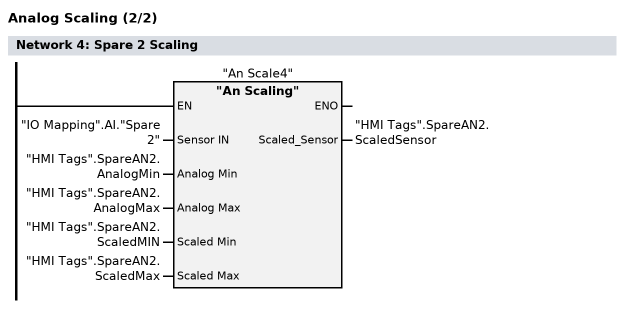
   RUNG wire#powerrail
      "An Scale4"("Sensor IN" := "IO Mapping".AI."Spare 2", "Analog Min" := "HMI Tags".SpareAN2.AnalogMin, "Analog Max" := "HMI Tags".SpareAN2.AnalogMax, "Scaled Min" := "HMI Tags".SpareAN2.ScaledMIN, "Scaled Max" := "HMI Tags".SpareAN2.ScaledMax, Scaled_Sensor => "HMI Tags".SpareAN2.ScaledSensor)
   END_RUNG
   // the same network as SCL:
   "An Scale4"("Sensor IN" := "IO Mapping".AI."Spare 2",   // "An Scaling"
               "Analog Min" := "HMI Tags".SpareAN2.AnalogMin,
               "Analog Max" := "HMI Tags".SpareAN2.AnalogMax,
               "Scaled Min" := "HMI Tags".SpareAN2.ScaledMIN,
               "Scaled Max" := "HMI Tags".SpareAN2.ScaledMax,
               Scaled_Sensor => "HMI Tags".SpareAN2.ScaledSensor);
END_REGION
END_FUNCTION

FUNCTION_BLOCK "An Scaling"   // FB5, LAD
{ S7_Optimized_Access := 'TRUE' }
// stored: MemoryReserve 100, SetENOAutomatically false
   VAR_INPUT
      "Sensor IN" : Int;
      "Analog Min" { ExternalAccessible := 'False'; ExternalVisible := 'False'; ExternalWritable := 'False'} : Int;
      "Analog Max" { ExternalAccessible := 'False'; ExternalVisible := 'False'; ExternalWritable := 'False'} : Int;
      "Scaled Min" { ExternalAccessible := 'False'; ExternalVisible := 'False'; ExternalWritable := 'False'} : Real;
      "Scaled Max" { ExternalAccessible := 'False'; ExternalVisible := 'False'; ExternalWritable := 'False'} : Real;
   END_VAR
   VAR_OUTPUT
      Scaled_Sensor : Real;
   END_VAR
   VAR
      Normalised_sensor { ExternalAccessible := 'False'; ExternalVisible := 'False'; ExternalWritable := 'False'} : Real;
      sensor_result { ExternalAccessible := 'False'; ExternalVisible := 'False'; ExternalWritable := 'False'} : Int;
   END_VAR
BEGIN

REGION Network 1: scale the sensor
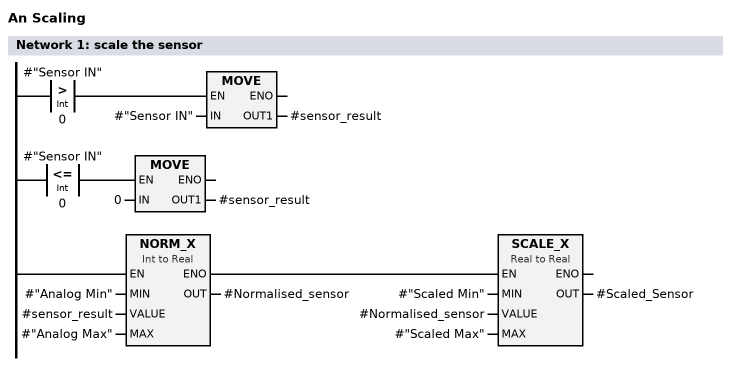
   RUNG wire#powerrail
      { S7_Templates := "SrcType := Int" } GT_Contact(in1 := #"Sensor IN", in2 := 0)
      { S7_GenerateENO := "TRUE" } Move(in := #"Sensor IN", out1 => #sensor_result)
   END_RUNG
   RUNG wire#powerrail
      { S7_Templates := "SrcType := Int" } LE_Contact(in1 := #"Sensor IN", in2 := 0)
      { S7_GenerateENO := "TRUE" } Move(in := 0, out1 => #sensor_result)
   END_RUNG
   RUNG wire#powerrail
      { S7_Templates := "[SrcType := Int, DestType := Real]"; S7_GenerateENO := "TRUE" } Normalize(min := #"Analog Min", value := #sensor_result, max := #"Analog Max", out => #Normalised_sensor)
      { S7_Templates := "[SrcType := Real, DestType := Real]"; S7_GenerateENO := "TRUE" } Scale(min := #"Scaled Min", value := #Normalised_sensor, max := #"Scaled Max", out => #Scaled_Sensor)
   END_RUNG
   // the same network as SCL:
   // ENO of a box is taken as its EN; it also drops when the box reports an error
   IF #"Sensor IN" > 0 THEN #sensor_result := #"Sensor IN"; END_IF;
   IF #"Sensor IN" <= 0 THEN #sensor_result := 0; END_IF;
   #Normalised_sensor := NORM_X(MIN := #"Analog Min", VALUE := #sensor_result, MAX := #"Analog Max");
   #Scaled_Sensor := SCALE_X(MIN := #"Scaled Min", VALUE := #Normalised_sensor, MAX := #"Scaled Max");
END_REGION
END_FUNCTION_BLOCK

FUNCTION "VFD Control" : Void   // FC9, LAD
{ S7_Optimized_Access := 'TRUE' }
// stored: SetENOAutomatically false
   VAR_TEMP   // added for the SCL form of the ladder/FBD networks
      _w1 : Bool;
   END_VAR
BEGIN

REGION Network 1: Liquids Pump
   // Refspeed = p2000, ref_Current = P2002, Ref_torque = P2003
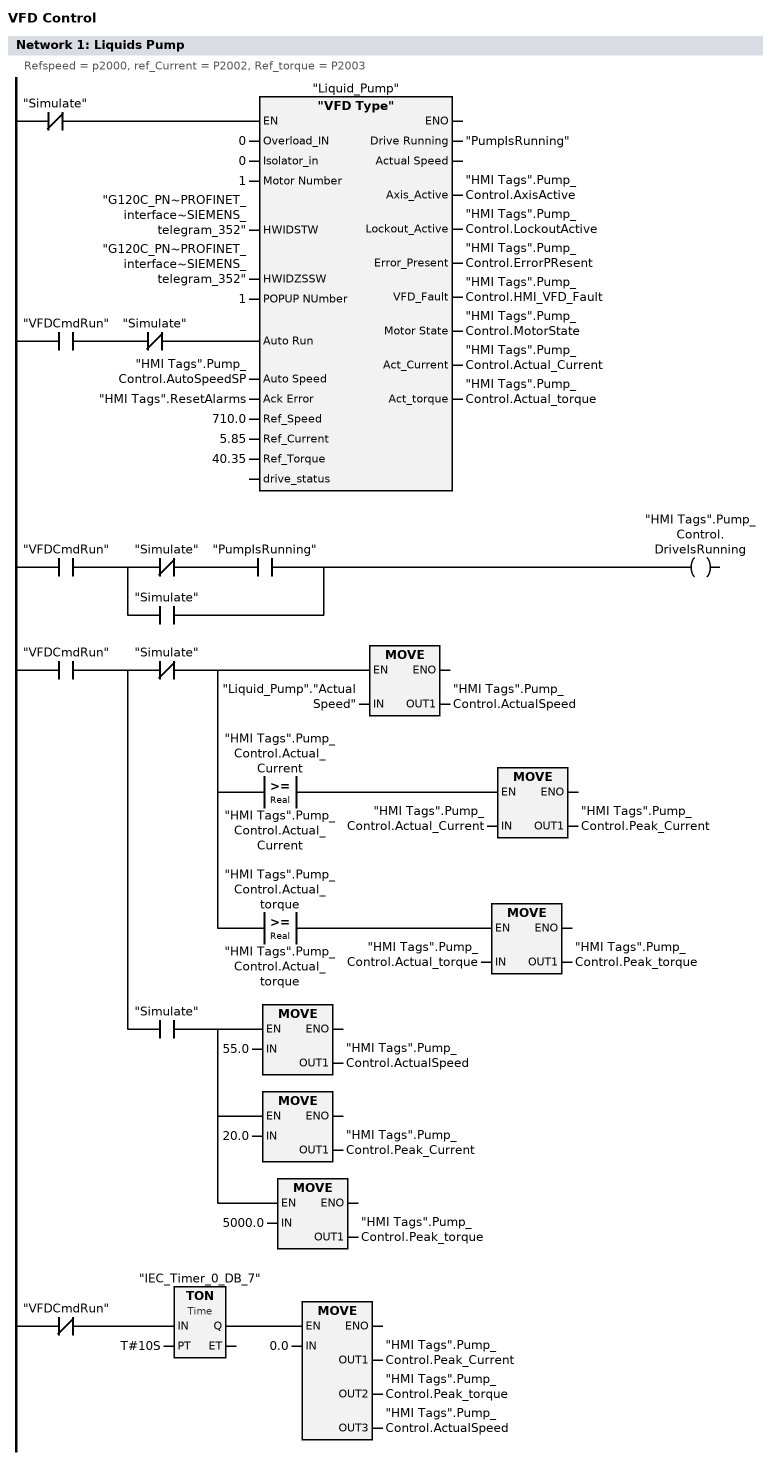
   RUNG wire#powerrail
      I_Contact( "Simulate" )
      "Liquid_Pump"("Auto Run" := wire#w1, Overload_IN := 0, Isolator_in := 0, "Motor Number" := 1, HWIDSTW := "G120C_PN~PROFINET_interface~SIEMENS_telegram_352", HWIDZSSW := "G120C_PN~PROFINET_interface~SIEMENS_telegram_352", "POPUP NUmber" := 1, "Auto Speed" := "HMI Tags".Pump_Control.AutoSpeedSP, "Ack Error" := "HMI Tags".ResetAlarms, Ref_Speed := 710.0, Ref_Current := 5.85, Ref_Torque := 40.35, drive_status :=, "Drive Running" => "PumpIsRunning", "Actual Speed" =>, Axis_Active => "HMI Tags".Pump_Control.AxisActive, Lockout_Active => "HMI Tags".Pump_Control.LockoutActive, Error_Present => "HMI Tags".Pump_Control.ErrorPResent, VFD_Fault => "HMI Tags".Pump_Control.HMI_VFD_Fault, "Motor State" => "HMI Tags".Pump_Control.MotorState, Act_Current => "HMI Tags".Pump_Control.Actual_Current, Act_torque => "HMI Tags".Pump_Control.Actual_torque)
   END_RUNG
   RUNG wire#powerrail
      Contact( "VFDCmdRun" )
      I_Contact( "Simulate" )
   END_RUNG wire#w1
   RUNG wire#powerrail
      Contact( "VFDCmdRun" )
      wire#w2
      I_Contact( "Simulate" )
      Contact( "PumpIsRunning" )
      wire#w3
      Coil( "HMI Tags".Pump_Control.DriveIsRunning )
   END_RUNG
   RUNG wire#w2
      Contact( "Simulate" )
   END_RUNG wire#w3
   RUNG wire#powerrail
      Contact( "VFDCmdRun" )
      wire#w4
      I_Contact( "Simulate" )
      wire#w5
      Move(in := "Liquid_Pump"."Actual Speed", out1 => "HMI Tags".Pump_Control.ActualSpeed)
   END_RUNG
   RUNG wire#w5
      { S7_Templates := "SrcType := Real" } GE_Contact(in1 := "HMI Tags".Pump_Control.Actual_Current, in2 := "HMI Tags".Pump_Control.Actual_Current)
      Move(in := "HMI Tags".Pump_Control.Actual_Current, out1 => "HMI Tags".Pump_Control.Peak_Current)
   END_RUNG
   RUNG wire#w5
      { S7_Templates := "SrcType := Real" } GE_Contact(in1 := "HMI Tags".Pump_Control.Actual_torque, in2 := "HMI Tags".Pump_Control.Actual_torque)
      Move(in := "HMI Tags".Pump_Control.Actual_torque, out1 => "HMI Tags".Pump_Control.Peak_torque)
   END_RUNG
   RUNG wire#w4
      Contact( "Simulate" )
      wire#w6
      Move(in := 55.0, out1 => "HMI Tags".Pump_Control.ActualSpeed)
   END_RUNG
   RUNG wire#w6
      Move(in := 20.0, out1 => "HMI Tags".Pump_Control.Peak_Current)
   END_RUNG
   RUNG wire#w6
      Move(in := 5000.0, out1 => "HMI Tags".Pump_Control.Peak_torque)
   END_RUNG
   RUNG wire#powerrail
      I_Contact( "VFDCmdRun" )
      { S7_Templates := "time_type := Time" } "IEC_Timer_0_DB_7".TON(pt := T#10S, et =>)
      Move(in := 0.0, out1 => "HMI Tags".Pump_Control.Peak_Current, out2 => "HMI Tags".Pump_Control.Peak_torque, out3 => "HMI Tags".Pump_Control.ActualSpeed)
   END_RUNG
   // the same network as SCL:
   IF NOT "Simulate" THEN
       "Liquid_Pump"(Overload_IN := 0,   // "VFD Type"
                     Isolator_in := 0,
                     "Motor Number" := 1,
                     HWIDSTW := "G120C_PN~PROFINET_interface~SIEMENS_telegram_352",
                     HWIDZSSW := "G120C_PN~PROFINET_interface~SIEMENS_telegram_352",
                     "POPUP NUmber" := 1,
                     "Auto Run" := "VFDCmdRun" AND NOT "Simulate",
                     "Auto Speed" := "HMI Tags".Pump_Control.AutoSpeedSP,
                     "Ack Error" := "HMI Tags".ResetAlarms,
                     Ref_Speed := 710.0,
                     Ref_Current := 5.85,
                     Ref_Torque := 40.35,
                     "Drive Running" => "PumpIsRunning",
                     Axis_Active => "HMI Tags".Pump_Control.AxisActive,
                     Lockout_Active => "HMI Tags".Pump_Control.LockoutActive,
                     Error_Present => "HMI Tags".Pump_Control.ErrorPResent,
                     VFD_Fault => "HMI Tags".Pump_Control.HMI_VFD_Fault,
                     "Motor State" => "HMI Tags".Pump_Control.MotorState,
                     Act_Current => "HMI Tags".Pump_Control.Actual_Current,
                     Act_torque => "HMI Tags".Pump_Control.Actual_torque);
   END_IF;
   "HMI Tags".Pump_Control.DriveIsRunning := "VFDCmdRun" AND ((NOT "Simulate" AND "PumpIsRunning") OR "Simulate");
   #_w1 := "VFDCmdRun" AND NOT "Simulate";
   IF #_w1 THEN "HMI Tags".Pump_Control.ActualSpeed := "Liquid_Pump"."Actual Speed"; END_IF;
   IF #_w1 AND ("HMI Tags".Pump_Control.Actual_Current >= "HMI Tags".Pump_Control.Actual_Current) THEN
       "HMI Tags".Pump_Control.Peak_Current := "HMI Tags".Pump_Control.Actual_Current;
   END_IF;
   IF #_w1 AND ("HMI Tags".Pump_Control.Actual_torque >= "HMI Tags".Pump_Control.Actual_torque) THEN
       "HMI Tags".Pump_Control.Peak_torque := "HMI Tags".Pump_Control.Actual_torque;
   END_IF;
   IF "VFDCmdRun" AND "Simulate" THEN
       "HMI Tags".Pump_Control.ActualSpeed := 55.0;
       "HMI Tags".Pump_Control.Peak_Current := 20.0;
       "HMI Tags".Pump_Control.Peak_torque := 5000.0;
   END_IF;
   "IEC_Timer_0_DB_7".TON(IN := NOT "VFDCmdRun", PT := T#10S);
   IF "IEC_Timer_0_DB_7".Q THEN
       "HMI Tags".Pump_Control.Peak_Current := 0.0;
       "HMI Tags".Pump_Control.Peak_torque := 0.0;
       "HMI Tags".Pump_Control.ActualSpeed := 0.0;
   END_IF;
END_REGION
END_FUNCTION

FUNCTION_BLOCK "VFD Type"   // FB9, LAD
{ S7_Optimized_Access := 'TRUE' }
// stored: MemoryReserve 100, SetENOAutomatically false
   VAR_INPUT
      Overload_IN { ExternalAccessible := 'False'; ExternalVisible := 'False'; ExternalWritable := 'False'} : Bool;
      Isolator_in { ExternalAccessible := 'False'; ExternalVisible := 'False'; ExternalWritable := 'False'} : Bool;
      "Motor Number" : Int;
      HWIDSTW { ExternalAccessible := 'False'; ExternalVisible := 'False'; ExternalWritable := 'False'} : HW_IO;
      HWIDZSSW { ExternalAccessible := 'False'; ExternalVisible := 'False'; ExternalWritable := 'False'} : HW_IO;
      "POPUP NUmber" : Int;
      "Auto Run" : Bool;
      "Auto Speed" : Real;
      "Ack Error" : Bool;
      Ref_Speed { ExternalAccessible := 'False'; ExternalVisible := 'False'; ExternalWritable := 'False'} : Real;
      Ref_Current : Real;
      Ref_Torque { ExternalAccessible := 'False'; ExternalVisible := 'False'; ExternalWritable := 'False'} : Real;
   END_VAR
   VAR_OUTPUT
      "Drive Running" : Bool;
      "Actual Speed" : Real;
      Axis_Active : Bool;
      Lockout_Active : Bool;
      Error_Present : Bool;
      VFD_Fault : Int;
      "Motor State" : Int;
      Act_Current : Real;
      Act_torque : Real;
   END_VAR
   VAR_IN_OUT
      drive_status { ExternalAccessible := 'False'; ExternalVisible := 'False'; ExternalWritable := 'False'} : Word;
   END_VAR
   VAR
      Speed_SP : Real;
      "Sts Running" : Bool;
   END_VAR
   VAR RETAIN
      IEC_Counter_0_Instance { ExternalAccessible := 'False'; ExternalVisible := 'False'; ExternalWritable := 'False'} : CTU_INT;
   END_VAR
   VAR
      "SCALED sp" : Real;
      "speed to drive" : Real;
      Speed_From_Drive : Real;
      "SCALED sp_1" : Real;
   END_VAR
BEGIN

REGION Network 1
   // Refspeed = p2000, ref_Current = P2002, Ref_torque = P2003
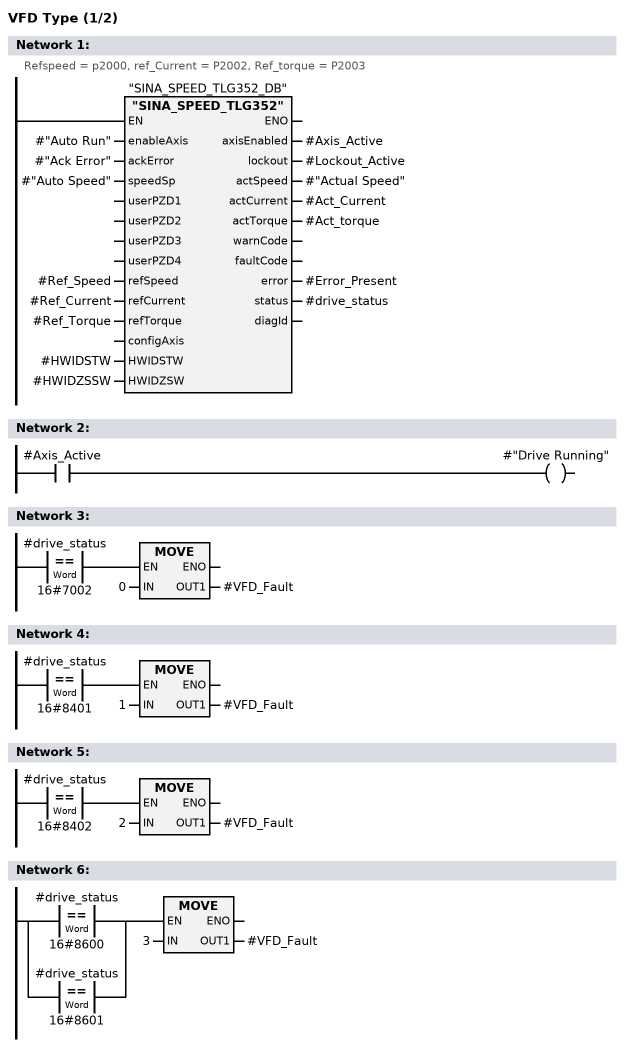
   RUNG wire#powerrail
      "SINA_SPEED_TLG352_DB"(enableAxis := #"Auto Run", ackError := #"Ack Error", speedSp := #"Auto Speed", userPZD1 :=, userPZD2 :=, userPZD3 :=, userPZD4 :=, refSpeed := #Ref_Speed, refCurrent := #Ref_Current, refTorque := #Ref_Torque, configAxis :=, HWIDSTW := #HWIDSTW, HWIDZSW := #HWIDZSSW, axisEnabled => #Axis_Active, lockout => #Lockout_Active, actSpeed => #"Actual Speed", actCurrent => #Act_Current, actTorque => #Act_torque, warnCode =>, faultCode =>, error => #Error_Present, status => #drive_status, diagId =>)
   END_RUNG
   // the same network as SCL:
   "SINA_SPEED_TLG352_DB"(enableAxis := #"Auto Run",   // "SINA_SPEED_TLG352"
                          ackError := #"Ack Error",
                          speedSp := #"Auto Speed",
                          refSpeed := #Ref_Speed,
                          refCurrent := #Ref_Current,
                          refTorque := #Ref_Torque,
                          HWIDSTW := #HWIDSTW,
                          HWIDZSW := #HWIDZSSW,
                          axisEnabled => #Axis_Active,
                          lockout => #Lockout_Active,
                          actSpeed => #"Actual Speed",
                          actCurrent => #Act_Current,
                          actTorque => #Act_torque,
                          error => #Error_Present,
                          status => #drive_status);
END_REGION

REGION Network 2
   RUNG wire#powerrail
      Contact( #Axis_Active )
      Coil( #"Drive Running" )
   END_RUNG
   // the same network as SCL:
   #"Drive Running" := #Axis_Active;
END_REGION

REGION Network 3
   RUNG wire#powerrail
      { S7_Templates := "SrcType := Word" } EQ_Contact(in1 := #drive_status, in2 := 16#7002)
      Move(in := 0, out1 => #VFD_Fault)
   END_RUNG
   // the same network as SCL:
   IF #drive_status = 16#7002 THEN #VFD_Fault := 0; END_IF;
END_REGION

REGION Network 4
   RUNG wire#powerrail
      { S7_Templates := "SrcType := Word" } EQ_Contact(in1 := #drive_status, in2 := 16#8401)
      Move(in := 1, out1 => #VFD_Fault)
   END_RUNG
   // the same network as SCL:
   IF #drive_status = 16#8401 THEN #VFD_Fault := 1; END_IF;
END_REGION

REGION Network 5
   RUNG wire#powerrail
      { S7_Templates := "SrcType := Word" } EQ_Contact(in1 := #drive_status, in2 := 16#8402)
      Move(in := 2, out1 => #VFD_Fault)
   END_RUNG
   // the same network as SCL:
   IF #drive_status = 16#8402 THEN #VFD_Fault := 2; END_IF;
END_REGION

REGION Network 6
   RUNG wire#powerrail
      { S7_Templates := "SrcType := Word" } EQ_Contact(in1 := #drive_status, in2 := 16#8600)
      wire#w1
      Move(in := 3, out1 => #VFD_Fault)
   END_RUNG
   RUNG wire#powerrail
      { S7_Templates := "SrcType := Word" } EQ_Contact(in1 := #drive_status, in2 := 16#8601)
   END_RUNG wire#w1
   // the same network as SCL:
   IF (#drive_status = 16#8600) OR (#drive_status = 16#8601) THEN #VFD_Fault := 3; END_IF;
END_REGION

REGION Network 7
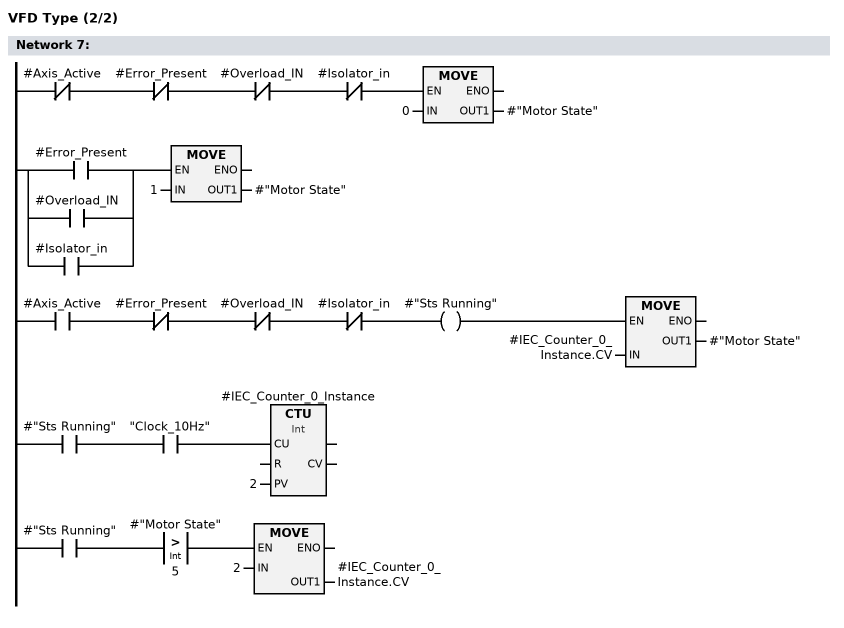
   RUNG wire#powerrail
      I_Contact( #Axis_Active )
      I_Contact( #Error_Present )
      I_Contact( #Overload_IN )
      I_Contact( #Isolator_in )
      Move(in := 0, out1 => #"Motor State")
   END_RUNG
   RUNG wire#powerrail
      Contact( #Error_Present )
      wire#w1
      Move(in := 1, out1 => #"Motor State")
   END_RUNG
   RUNG wire#powerrail
      Contact( #Overload_IN )
   END_RUNG wire#w1
   RUNG wire#powerrail
      Contact( #Isolator_in )
   END_RUNG wire#w1
   RUNG wire#powerrail
      Contact( #Axis_Active )
      I_Contact( #Error_Present )
      I_Contact( #Overload_IN )
      I_Contact( #Isolator_in )
      Coil( #"Sts Running" )
      Move(in := #IEC_Counter_0_Instance.CV, out1 => #"Motor State")
   END_RUNG
   RUNG wire#powerrail
      Contact( #"Sts Running" )
      Contact( "Clock_10Hz" )
      { S7_Templates := "value_type := Int" } #IEC_Counter_0_Instance.CTU(r :=, pv := 2, cv =>)
   END_RUNG
   RUNG wire#powerrail
      Contact( #"Sts Running" )
      { S7_Templates := "SrcType := Int" } GT_Contact(in1 := #"Motor State", in2 := 5)
      Move(in := 2, out1 => #IEC_Counter_0_Instance.CV)
   END_RUNG
   // the same network as SCL:
   IF NOT #Axis_Active AND NOT #Error_Present AND NOT #Overload_IN AND NOT #Isolator_in THEN
       #"Motor State" := 0;
   END_IF;
   IF #Error_Present OR #Overload_IN OR #Isolator_in THEN #"Motor State" := 1; END_IF;
   #"Sts Running" := #Axis_Active AND NOT #Error_Present AND NOT #Overload_IN AND NOT #Isolator_in;
   IF #"Sts Running" THEN #"Motor State" := #IEC_Counter_0_Instance.CV; END_IF;
   #IEC_Counter_0_Instance(CU := #"Sts Running" AND "Clock_10Hz", PV := 2);   // CTU
   IF #"Sts Running" AND (#"Motor State" > 5) THEN #IEC_Counter_0_Instance.CV := 2; END_IF;
END_REGION
END_FUNCTION_BLOCK

FUNCTION_BLOCK "SINA_SPEED_TLG352"
TITLE = Speed control S7 to SINAMICS using Standardtelegram 352
{ S7_Optimized_Access := 'TRUE' }
AUTHOR : SIEMENS
FAMILY : DRIVES
NAME : SINA_SPD_TLG352
VERSION : 1.0
//The function block SINA_SPEED_TLG352 controls a SINAMICS drive using SIEMENS telegram 352
   VAR_INPUT 
      enableAxis : Bool;   // 0 -> 1 = Enable the drive (OFF2 / OFF 3 are 1 in default status) (OFF1 = 0->1)
      ackError : Bool;   // 0 -> 1 = Acknowledge drive error
      speedSp : Real;   // Speed setpoint [rpm]
      userPZD1 : Word;   // User PZD1
      userPZD2 : Word;   // User PZD2
      userPZD3 : Word;   // User PZD3
      userPZD4 : Word;   // User PZD4
      refSpeed : Real;   // Reference speed [p2000] in [rpm]
      refCurrent : Real;   // Reference current [p2002] in [Aeff]
      refTorque : Real;   // Reference torque [p2003] in [Nm]
      configAxis : Word := 16#003F;   // binary programmed input to control all functions in the telegram without its own function block input
      HWIDSTW : HW_IO;   // Hardware Identifer set point slot
      HWIDZSW : HW_IO;   // Hardware Identifer actual value slot
   END_VAR

   VAR_OUTPUT 
      axisEnabled : Bool;   // 1 = Drive is enabled
      lockout : Bool;   // 1 = Drive lockout active
      actSpeed : Real;   // Smoothed actual speed in [1/min]
      actCurrent : Real;   // Smoothed current actual in [Arms]
      actTorque : Real;   // Actual smoothed torque in [Nm]
      warnCode : UInt;   // Warn code of the drive
      faultCode : UInt;   // Fault code of the drive
      error : Bool;   // 1 = Error (FB and Infeed)
      status : Int;   // Status output (7002 = FB in operation; 7xxx = warning; 8xxx = error description - read the manual)
      diagId : Int;   // Error codes of the system function blocks DPWR / DPRD_DAT
   END_VAR

   VAR_TEMP 
      tempSpeed : Real;   // Speed setpoint in percent
      tempRefValueInvalid : Bool;   // At least one reference value is or < 0
      tempSendBuf : Array[0..5] of Word;   // Send buffer
      tempRecvBuf : Array[0..5] of Word;   // Receive buffer
   END_VAR

   VAR CONSTANT 
      NORMALIZATION_VALUE : Int := 16#4000;   // Used to calculate the Real values
      MAX_INT : Int := 16#7FFF;
      MIN_INT : Int := 16#8000;
      NO_ERROR : Int := 16#7002;   // No error
      REF_CURRRENT_INVALID : Int := 16#7010;   // RefCurrent input is 0 or < 0
      REF_TORQUE_INVALID : Int := 16#7011;   // RefTorque input is 0 or < 0
      REF_VALUES_INVALID : Int := 16#7013;   // Multiple reference values are 0 or < 0
      WARNING_WARN_CODE : Int := 16#7005;   // warnCode is not 0
      REF_SPEED_INVALID : Int := 16#8001;   // RefSpeed input is 0 or < 0
      ERROR_DRIVE : Int := 16#8401;   // Drive error
      ERROR_LOCKOUT : Int := 16#8402;   // Drive lockout
      ERROR_DPREAD : Int := 16#8600;   // DPRD_DAT returned an error
      ERROR_DPWRITE : Int := 16#8601;   // DPWR_DAT returned an error
      ERROR_FAULT_CODE : Int := 16#8800;   // faultCode is not 0
      STW1 : USInt := 0;
      ZSW1 : USInt := 0;
      NSOLL_A : USInt := 1;
   END_VAR


BEGIN
	//=============================================================================
	//SIEMENS AG
	//(c)Copyright 2019 All Rights Reserved
	//-----------------------------------------------------------------------------
	// Library:       LSINAExt
	// Tested with:   SIMATIC S7 CPU 1513-1 PN V2.5
	// Engineering:   TIA Portal V15
	// Restrictions:  -
	// Requirements:  S7-1200 / S7-1500
	// Functionality: cyclic communication between a SINAMICS a PLC.
	//                If in HWConfig SIEMENS telegram 352 are projected 6 PZD-words are exchanged
	//                in every bus cycle.
	//                The parametrisation of these words is described in the manual of the
	//                SINAMICS
	//-----------------------------------------------------------------------------
	//Change log table:
	//Version  Date       Expert in charge Changes applied
	//01.00.00 11.02.2019 (AS) First released version
	//=============================================================================
	
	// Prepare PZD1 (STW1)
	#tempSendBuf[#STW1].%X0 := #enableAxis;
	#tempSendBuf[#STW1].%X7 := #ackError;
	#tempSendBuf[#STW1].%X1 := #configAxis.%X0;
	#tempSendBuf[#STW1].%X2 := #configAxis.%X1;
	#tempSendBuf[#STW1].%X3 := #configAxis.%X2;
	#tempSendBuf[#STW1].%X4 := #configAxis.%X3;
	#tempSendBuf[#STW1].%X5 := #configAxis.%X4;
	#tempSendBuf[#STW1].%X6 := #configAxis.%X5;
	#tempSendBuf[#STW1].%X11 := #configAxis.%X6;
	#tempSendBuf[#STW1].%X13 := #configAxis.%X7;
	#tempSendBuf[#STW1].%X14 := #configAxis.%X8;
	#tempSendBuf[#STW1].%X10 := TRUE; // control by PLC
	
	// Speed
	IF #refSpeed > 0 THEN
	    #tempSpeed := #speedSp * (#NORMALIZATION_VALUE / #refSpeed);
	    // Limit REAL - Variable to INT - limits
	    IF #tempSpeed > #MAX_INT THEN
	        #tempSpeed := #MAX_INT;
	    ELSIF #tempSpeed < #MIN_INT THEN
	        #tempSpeed := #MIN_INT;
	    ELSE
	        ; // not needed
	    END_IF;
	    #tempSendBuf[#NSOLL_A] := INT_TO_WORD(REAL_TO_INT(#tempSpeed));
	ELSE
	    #error := TRUE;
	    #status := #REF_SPEED_INVALID;
	    #tempSendBuf[#NSOLL_A] := W#16#0;
	END_IF;
	
	#tempSendBuf[2] := #userPZD1;
	#tempSendBuf[3] := #userPZD2;
	#tempSendBuf[4] := #userPZD3;
	#tempSendBuf[5] := #userPZD4;
	
	// Send telegram to drive
	#diagId := DPWR_DAT(LADDR := #HWIDSTW,
	                    RECORD := #tempSendBuf);
	
	// Error when writing the telegram
	IF #diagId <> 0 THEN
	    #error := TRUE;
	    #status := #ERROR_DPWRITE;
	    
	    // Reset outputs
	    #actSpeed := 0.0;
	    #actCurrent := 0.0;
	    #actTorque := 0.0;
	    #warnCode := 0;
	    #faultCode := 0;
	    
	    RETURN;
	ELSE
	    ;
	END_IF;
	
	// Receive telegram from drive
	#diagId := DPRD_DAT(LADDR := #HWIDZSW,
	                    RECORD => #tempRecvBuf);
	
	// Error when reading the telegram
	IF #diagId <> 0 THEN
	    #error := TRUE;
	    #status := #ERROR_DPREAD;
	    
	    // Reset outputs
	    #actSpeed := 0.0;
	    #actCurrent := 0.0;
	    #actTorque := 0.0;
	    #warnCode := 0;
	    #faultCode := 0;
	    
	    RETURN;
	ELSE
	    ;
	END_IF;
	
	// Analyse ZSW1
	#axisEnabled := #tempRecvBuf[#ZSW1].%X2;
	#lockout := #tempRecvBuf[#ZSW1].%X6;
	#error := #tempRecvBuf[#ZSW1].%X3 OR #tempRecvBuf[#ZSW1].%X6;
	
	IF #tempRecvBuf[#ZSW1].%X3 THEN
	    #status := #ERROR_DRIVE;
	ELSIF #tempRecvBuf[#ZSW1].%X6 THEN
	    #status := #ERROR_LOCKOUT;
	ELSE
	    #status := #NO_ERROR;
	END_IF;
	
	// Actual speed
	IF (#refSpeed <= 0)
	    AND #enableAxis
	THEN
	    #actSpeed := 0.0;
	    #error := TRUE;
	    #status := #REF_SPEED_INVALID;
	ELSE
	    #actSpeed := INT_TO_REAL(WORD_TO_INT(#tempRecvBuf[1])) / (#NORMALIZATION_VALUE / #refSpeed);
	END_IF;
	
	// Actual current
	IF (#refCurrent <= 0)
	    AND #enableAxis
	    AND NOT #error
	THEN
	    #actCurrent := 0.0;
	    
	    IF #tempRefValueInvalid THEN
	        #status := #REF_VALUES_INVALID;
	    ELSE
	        #status := #REF_CURRRENT_INVALID;
	        #tempRefValueInvalid := TRUE;
	    END_IF;
	ELSE
	    #actCurrent := INT_TO_REAL(WORD_TO_INT(#tempRecvBuf[2])) / (#NORMALIZATION_VALUE / #refCurrent);
	END_IF;
	
	// Actual torque
	IF (#refTorque <= 0)
	    AND #enableAxis
	    AND NOT #error
	THEN
	    #actTorque := 0.0;
	    
	    IF #tempRefValueInvalid THEN
	        #status := #REF_VALUES_INVALID;
	    ELSE
	        #status := #REF_TORQUE_INVALID;
	        #tempRefValueInvalid := TRUE;
	    END_IF;
	ELSE
	    #actTorque := INT_TO_REAL(WORD_TO_INT(#tempRecvBuf[3])) / (#NORMALIZATION_VALUE / #refTorque);
	END_IF;
	
	// Warn code
	#warnCode := WORD_TO_UINT(#tempRecvBuf[4]);
	IF #warnCode <> 0
	    AND NOT #error
	THEN
	    #status := #WARNING_WARN_CODE;
	ELSE
	    ;
	END_IF;
	
	// Fault code
	#faultCode := WORD_TO_UINT(#tempRecvBuf[5]);
	IF #faultCode <> 0 THEN
	    #error := TRUE;
	    #status := #ERROR_FAULT_CODE;
	ELSE
	    ;
	END_IF;
END_FUNCTION_BLOCK

FUNCTION "Flowmeter Diag" : Void   // FC10, LAD
{ S7_Optimized_Access := 'TRUE' }
// stored: SetENOAutomatically false
BEGIN

REGION Network 1
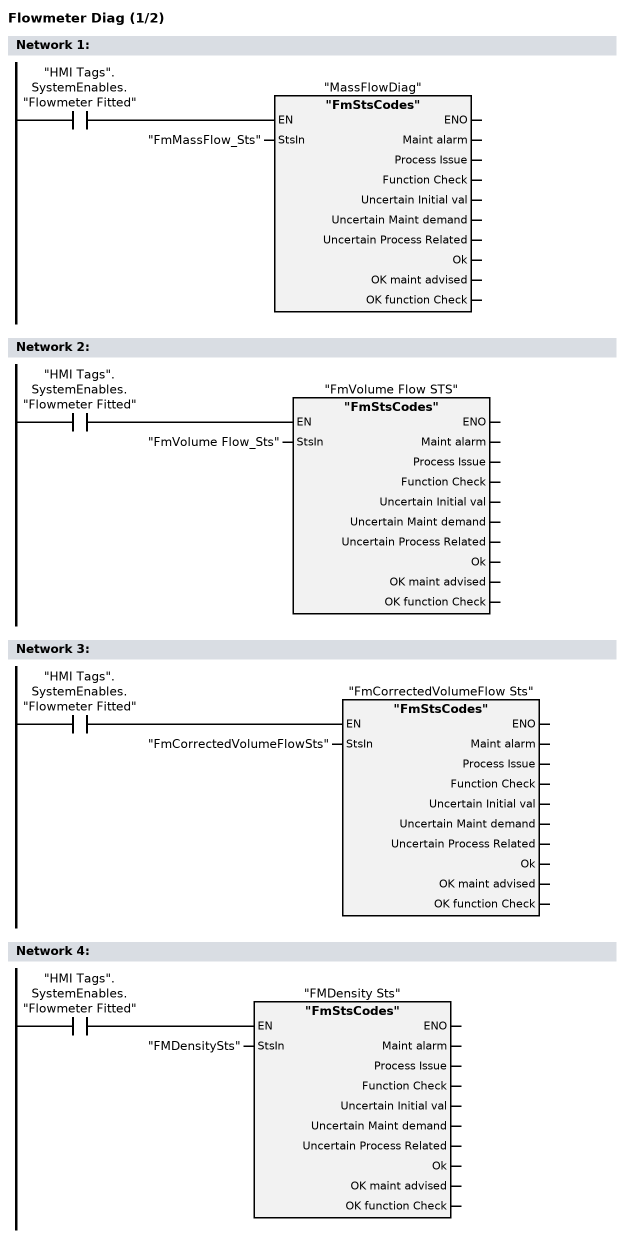
   RUNG wire#powerrail
      Contact( "HMI Tags".SystemEnables."Flowmeter Fitted" )
      "MassFlowDiag"(StsIn := "FmMassFlow_Sts", "Maint alarm" =>, "Process Issue" =>, "Function Check" =>, "Uncertain Initial val" =>, "Uncertain Maint demand" =>, "Uncertain Process Related" =>, Ok =>, "OK maint advised" =>, "OK function Check" =>)
   END_RUNG
   // the same network as SCL:
   IF "HMI Tags".SystemEnables."Flowmeter Fitted" THEN
       "MassFlowDiag"(StsIn := "FmMassFlow_Sts");   // "FmStsCodes"
   END_IF;
END_REGION

REGION Network 2
   RUNG wire#powerrail
      Contact( "HMI Tags".SystemEnables."Flowmeter Fitted" )
      "FmVolume Flow STS"(StsIn := "FmVolume Flow_Sts", "Maint alarm" =>, "Process Issue" =>, "Function Check" =>, "Uncertain Initial val" =>, "Uncertain Maint demand" =>, "Uncertain Process Related" =>, Ok =>, "OK maint advised" =>, "OK function Check" =>)
   END_RUNG
   // the same network as SCL:
   IF "HMI Tags".SystemEnables."Flowmeter Fitted" THEN
       "FmVolume Flow STS"(StsIn := "FmVolume Flow_Sts");   // "FmStsCodes"
   END_IF;
END_REGION

REGION Network 3
   RUNG wire#powerrail
      Contact( "HMI Tags".SystemEnables."Flowmeter Fitted" )
      "FmCorrectedVolumeFlow Sts"(StsIn := "FmCorrectedVolumeFlowSts", "Maint alarm" =>, "Process Issue" =>, "Function Check" =>, "Uncertain Initial val" =>, "Uncertain Maint demand" =>, "Uncertain Process Related" =>, Ok =>, "OK maint advised" =>, "OK function Check" =>)
   END_RUNG
   // the same network as SCL:
   IF "HMI Tags".SystemEnables."Flowmeter Fitted" THEN
       "FmCorrectedVolumeFlow Sts"(StsIn := "FmCorrectedVolumeFlowSts");   // "FmStsCodes"
   END_IF;
END_REGION

REGION Network 4
   RUNG wire#powerrail
      Contact( "HMI Tags".SystemEnables."Flowmeter Fitted" )
      "FMDensity Sts"(StsIn := "FMDensitySts", "Maint alarm" =>, "Process Issue" =>, "Function Check" =>, "Uncertain Initial val" =>, "Uncertain Maint demand" =>, "Uncertain Process Related" =>, Ok =>, "OK maint advised" =>, "OK function Check" =>)
   END_RUNG
   // the same network as SCL:
   IF "HMI Tags".SystemEnables."Flowmeter Fitted" THEN
       "FMDensity Sts"(StsIn := "FMDensitySts");   // "FmStsCodes"
   END_IF;
END_REGION

REGION Network 5
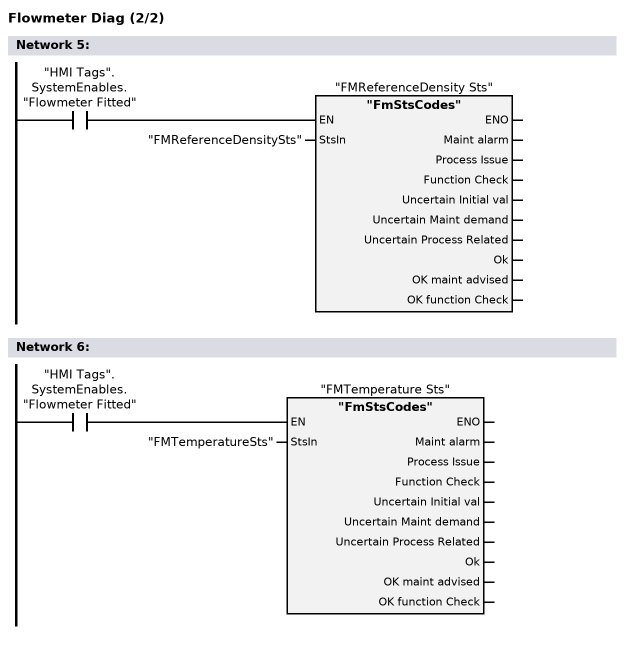
   RUNG wire#powerrail
      Contact( "HMI Tags".SystemEnables."Flowmeter Fitted" )
      "FMReferenceDensity Sts"(StsIn := "FMReferenceDensitySts", "Maint alarm" =>, "Process Issue" =>, "Function Check" =>, "Uncertain Initial val" =>, "Uncertain Maint demand" =>, "Uncertain Process Related" =>, Ok =>, "OK maint advised" =>, "OK function Check" =>)
   END_RUNG
   // the same network as SCL:
   IF "HMI Tags".SystemEnables."Flowmeter Fitted" THEN
       "FMReferenceDensity Sts"(StsIn := "FMReferenceDensitySts");   // "FmStsCodes"
   END_IF;
END_REGION

REGION Network 6
   RUNG wire#powerrail
      Contact( "HMI Tags".SystemEnables."Flowmeter Fitted" )
      "FMTemperature Sts"(StsIn := "FMTemperatureSts", "Maint alarm" =>, "Process Issue" =>, "Function Check" =>, "Uncertain Initial val" =>, "Uncertain Maint demand" =>, "Uncertain Process Related" =>, Ok =>, "OK maint advised" =>, "OK function Check" =>)
   END_RUNG
   // the same network as SCL:
   IF "HMI Tags".SystemEnables."Flowmeter Fitted" THEN
       "FMTemperature Sts"(StsIn := "FMTemperatureSts");   // "FmStsCodes"
   END_IF;
END_REGION
END_FUNCTION

FUNCTION_BLOCK "FmStsCodes"   // FB2, LAD
{ S7_Optimized_Access := 'TRUE' }
// stored: MemoryReserve 100, SetENOAutomatically false
   VAR_INPUT
      StsIn : Byte;
   END_VAR
   VAR_OUTPUT
      "Maint alarm" : Bool;
      "Process Issue" : Bool;
      "Function Check" : Bool;
      "Uncertain Initial val" : Bool;
      "Uncertain Maint demand" : Bool;
      "Uncertain Process Related" : Bool;
      Ok : Bool;
      "OK maint advised" : Bool;
      "OK function Check" : Bool;
   END_VAR
   VAR
      Val1 : Byte;
   END_VAR
BEGIN

REGION Network 1: 0x24 = 36 BAD maintenance alarm
   // A measured value is not available because a device
   // error has occurred
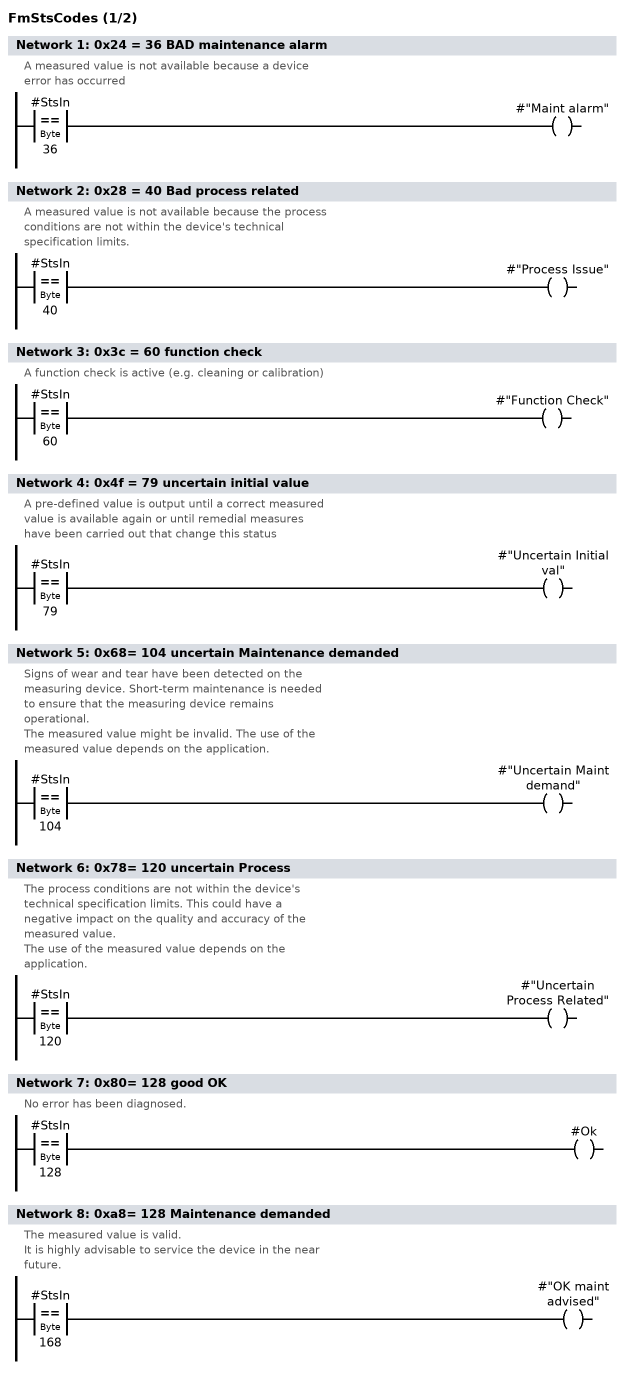
   RUNG wire#powerrail
      { S7_Templates := "SrcType := Byte" } EQ_Contact(in1 := #StsIn, in2 := 36)
      Coil( #"Maint alarm" )
   END_RUNG
   // the same network as SCL:
   #"Maint alarm" := #StsIn = 36;
END_REGION

REGION Network 2: 0x28 = 40 Bad process related
   // A measured value is not available because the process
   // conditions are not within the device's technical
   // specification limits.
   RUNG wire#powerrail
      { S7_Templates := "SrcType := Byte" } EQ_Contact(in1 := #StsIn, in2 := 40)
      Coil( #"Process Issue" )
   END_RUNG
   // the same network as SCL:
   #"Process Issue" := #StsIn = 40;
END_REGION

REGION Network 3: 0x3c = 60 function check
   // A function check is active (e.g. cleaning or calibration)
   RUNG wire#powerrail
      { S7_Templates := "SrcType := Byte" } EQ_Contact(in1 := #StsIn, in2 := 60)
      Coil( #"Function Check" )
   END_RUNG
   // the same network as SCL:
   #"Function Check" := #StsIn = 60;
END_REGION

REGION Network 4: 0x4f = 79 uncertain initial value
   // A pre-defined value is output until a correct measured
   // value is available again or until remedial measures
   // have been carried out that change this status
   RUNG wire#powerrail
      { S7_Templates := "SrcType := Byte" } EQ_Contact(in1 := #StsIn, in2 := 79)
      Coil( #"Uncertain Initial val" )
   END_RUNG
   // the same network as SCL:
   #"Uncertain Initial val" := #StsIn = 79;
END_REGION

REGION Network 5: 0x68= 104 uncertain Maintenance demanded
   // Signs of wear and tear have been detected on the
   // measuring device. Short-term maintenance is needed
   // to ensure that the measuring device remains
   // operational.
   // The measured value might be invalid. The use of the
   // measured value depends on the application.
   RUNG wire#powerrail
      { S7_Templates := "SrcType := Byte" } EQ_Contact(in1 := #StsIn, in2 := 104)
      Coil( #"Uncertain Maint demand" )
   END_RUNG
   // the same network as SCL:
   #"Uncertain Maint demand" := #StsIn = 104;
END_REGION

REGION Network 6: 0x78= 120 uncertain Process
   // The process conditions are not within the device's
   // technical specification limits. This could have a
   // negative impact on the quality and accuracy of the
   // measured value.
   // The use of the measured value depends on the
   // application.
   RUNG wire#powerrail
      { S7_Templates := "SrcType := Byte" } EQ_Contact(in1 := #StsIn, in2 := 120)
      Coil( #"Uncertain Process Related" )
   END_RUNG
   // the same network as SCL:
   #"Uncertain Process Related" := #StsIn = 120;
END_REGION

REGION Network 7: 0x80= 128 good OK
   // No error has been diagnosed.
   RUNG wire#powerrail
      { S7_Templates := "SrcType := Byte" } EQ_Contact(in1 := #StsIn, in2 := 128)
      Coil( #Ok )
   END_RUNG
   // the same network as SCL:
   #Ok := #StsIn = 128;
END_REGION

REGION Network 8: 0xa8= 128 Maintenance demanded
   // The measured value is valid.
   // It is highly advisable to service the device in the near
   // future.
   RUNG wire#powerrail
      { S7_Templates := "SrcType := Byte" } EQ_Contact(in1 := #StsIn, in2 := 168)
      Coil( #"OK maint advised" )
   END_RUNG
   // the same network as SCL:
   #"OK maint advised" := #StsIn = 168;
END_REGION

REGION Network 9: 0xbc= 188 GOOD - Function check
   // The measured value is valid.
   // The measuring device is performing an internal
   // function check. The function check does not have any
   // noticeable effect on the process.
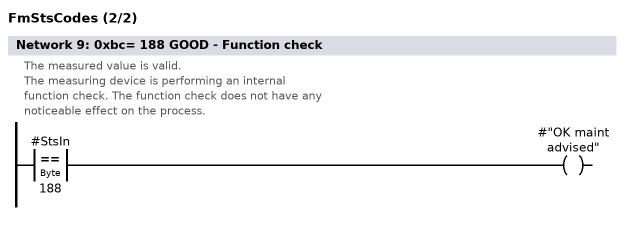
   RUNG wire#powerrail
      { S7_Templates := "SrcType := Byte" } EQ_Contact(in1 := #StsIn, in2 := 188)
      Coil( #"OK maint advised" )
   END_RUNG
   // the same network as SCL:
   #"OK maint advised" := #StsIn = 188;
END_REGION
END_FUNCTION_BLOCK

FUNCTION_BLOCK "GBL_TandD"   // FB20, LAD
{ S7_Optimized_Access := 'TRUE' }
// stored: MemoryReserve 100, SetENOAutomatically false
   VAR
      "write time" { ExternalAccessible := 'False'; ExternalVisible := 'False'; ExternalWritable := 'False'} : DTL;
      "System Time" { ExternalAccessible := 'False'; ExternalVisible := 'False'; ExternalWritable := 'False'} : DTL;
   END_VAR
   VAR_TEMP   // added for the SCL form of the ladder/FBD networks
      _w1 : Bool;
   END_VAR
BEGIN

REGION Network 1
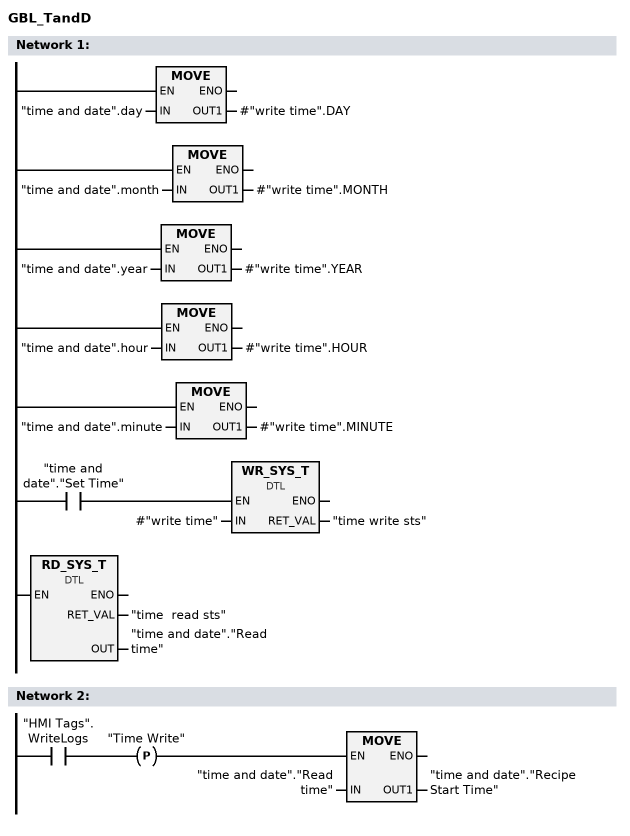
   RUNG wire#powerrail
      Move(in := "time and date".day, out1 => #"write time".DAY)
   END_RUNG
   RUNG wire#powerrail
      Move(in := "time and date".month, out1 => #"write time".MONTH)
   END_RUNG
   RUNG wire#powerrail
      Move(in := "time and date".year, out1 => #"write time".YEAR)
   END_RUNG
   RUNG wire#powerrail
      Move(in := "time and date".hour, out1 => #"write time".HOUR)
   END_RUNG
   RUNG wire#powerrail
      Move(in := "time and date".minute, out1 => #"write time".MINUTE)
   END_RUNG
   RUNG wire#powerrail
      Contact( "time and date"."Set Time" )
      { S7_Templates := "date_type := DTL" } WR_SYS_T(IN := #"write time", RET_VAL => "time write sts")
   END_RUNG
   RUNG wire#powerrail
      { S7_Templates := "date_type := DTL" } RD_SYS_T(RET_VAL => "time  read sts", OUT => "time and date"."Read time")
   END_RUNG
   // the same network as SCL:
   #"write time".DAY := "time and date".day;
   #"write time".MONTH := "time and date".month;
   #"write time".YEAR := "time and date".year;
   #"write time".HOUR := "time and date".hour;
   #"write time".MINUTE := "time and date".minute;
   IF "time and date"."Set Time" THEN "time write sts" := WR_SYS_T(IN := #"write time"); END_IF;
   "time  read sts" := RD_SYS_T(OUT => "time and date"."Read time");
END_REGION

REGION Network 2
   RUNG wire#powerrail
      Contact( "HMI Tags".WriteLogs )
      P_Trig( "Time Write" )
      Move(in := "time and date"."Read time", out1 => "time and date"."Recipe Start Time")
   END_RUNG
   // the same network as SCL:
   #_w1 := "HMI Tags".WriteLogs AND NOT "Time Write";   // rising edge
   "Time Write" := "HMI Tags".WriteLogs;
   IF #_w1 THEN "time and date"."Recipe Start Time" := "time and date"."Read time"; END_IF;
END_REGION
END_FUNCTION_BLOCK

FUNCTION "Assign_Output" : Void   // FC6, LAD
{ S7_Optimized_Access := 'TRUE' }
// stored: SetENOAutomatically false
   VAR_INPUT
      Out : Bool;
      outputSelection : Int;
   END_VAR
   VAR_OUTPUT
      output1 : Bool;
      output2 : Bool;
      output3 : Bool;
      output4 : Bool;
      output5 : Bool;
      output6 : Bool;
      output7 : Bool;
      output8 : Bool;
      output9 : Bool;
      output10 : Bool;
      outputSelected : Int;
   END_VAR
BEGIN

REGION Network 1
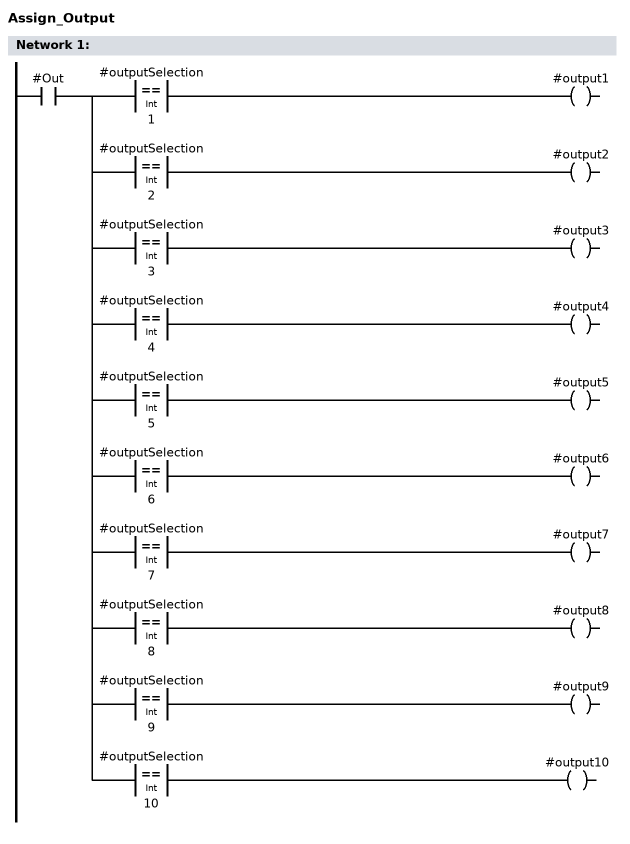
   RUNG wire#powerrail
      Contact( #Out )
      wire#w1
      { S7_Templates := "SrcType := Int" } EQ_Contact(in1 := #outputSelection, in2 := 1)
      Coil( #output1 )
   END_RUNG
   RUNG wire#w1
      { S7_Templates := "SrcType := Int" } EQ_Contact(in1 := #outputSelection, in2 := 2)
      Coil( #output2 )
   END_RUNG
   RUNG wire#w1
      { S7_Templates := "SrcType := Int" } EQ_Contact(in1 := #outputSelection, in2 := 3)
      Coil( #output3 )
   END_RUNG
   RUNG wire#w1
      { S7_Templates := "SrcType := Int" } EQ_Contact(in1 := #outputSelection, in2 := 4)
      Coil( #output4 )
   END_RUNG
   RUNG wire#w1
      { S7_Templates := "SrcType := Int" } EQ_Contact(in1 := #outputSelection, in2 := 5)
      Coil( #output5 )
   END_RUNG
   RUNG wire#w1
      { S7_Templates := "SrcType := Int" } EQ_Contact(in1 := #outputSelection, in2 := 6)
      Coil( #output6 )
   END_RUNG
   RUNG wire#w1
      { S7_Templates := "SrcType := Int" } EQ_Contact(in1 := #outputSelection, in2 := 7)
      Coil( #output7 )
   END_RUNG
   RUNG wire#w1
      { S7_Templates := "SrcType := Int" } EQ_Contact(in1 := #outputSelection, in2 := 8)
      Coil( #output8 )
   END_RUNG
   RUNG wire#w1
      { S7_Templates := "SrcType := Int" } EQ_Contact(in1 := #outputSelection, in2 := 9)
      Coil( #output9 )
   END_RUNG
   RUNG wire#w1
      { S7_Templates := "SrcType := Int" } EQ_Contact(in1 := #outputSelection, in2 := 10)
      Coil( #output10 )
   END_RUNG
   // the same network as SCL:
   #output1 := #Out AND (#outputSelection = 1);
   #output2 := #Out AND (#outputSelection = 2);
   #output3 := #Out AND (#outputSelection = 3);
   #output4 := #Out AND (#outputSelection = 4);
   #output5 := #Out AND (#outputSelection = 5);
   #output6 := #Out AND (#outputSelection = 6);
   #output7 := #Out AND (#outputSelection = 7);
   #output8 := #Out AND (#outputSelection = 8);
   #output9 := #Out AND (#outputSelection = 9);
   #output10 := #Out AND (#outputSelection = 10);
END_REGION
END_FUNCTION

FUNCTION_BLOCK "Pressure Type"   // FB11, LAD
{ S7_Optimized_Access := 'TRUE' }
// stored: MemoryReserve 100, SetENOAutomatically false
   VAR_INPUT
      "RAW INPUT" : Int;
      "Scale MIN" : Real;
      "Scale MAX" : Real;
   END_VAR
   VAR_OUTPUT
      PV : Real;
   END_VAR
   VAR
      IEC_Timer_0_Instance_2 { S7_SetPoint := 'True'} : TON_TIME;
      IEC_Timer_0_Instance { S7_SetPoint := 'True'} : TOF_TIME;
      "INT TO REAL" { ExternalAccessible := 'False'; ExternalVisible := 'False'; ExternalWritable := 'False'} : Real;
      "DINT TO REAL" { ExternalAccessible := 'False'; ExternalVisible := 'False'; ExternalWritable := 'False'} : Real;
   END_VAR
   VAR CONSTANT
      "0" : Int := 0;
      "1" : Int := 1;
   END_VAR
BEGIN

REGION Network 1
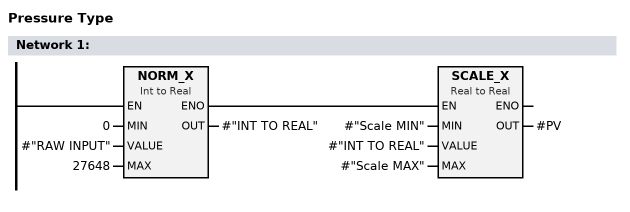
   RUNG wire#powerrail
      { S7_Templates := "[SrcType := Int, DestType := Real]" } Normalize(min := 0, value := #"RAW INPUT", max := 27648, out => #"INT TO REAL")
      { S7_Templates := "[SrcType := Real, DestType := Real]" } Scale(min := #"Scale MIN", value := #"INT TO REAL", max := #"Scale MAX", out => #PV)
   END_RUNG
   // the same network as SCL:
   #"INT TO REAL" := NORM_X(MIN := 0, VALUE := #"RAW INPUT", MAX := 27648);
   #PV := SCALE_X(MIN := #"Scale MIN", VALUE := #"INT TO REAL", MAX := #"Scale MAX");
END_REGION
END_FUNCTION_BLOCK

FUNCTION_BLOCK "Temperature Type"   // FB4, LAD
{ S7_Optimized_Access := 'TRUE' }
// stored: MemoryReserve 100, SetENOAutomatically false
   VAR_INPUT
      "RAW INPUT" : Int;
      "Scale MIN" : Real;
      "Scale MAX" : Real;
   END_VAR
   VAR_OUTPUT
      PV : Real;
   END_VAR
   VAR
      IEC_Timer_0_Instance_2 { S7_SetPoint := 'True'} : TON_TIME;
      IEC_Timer_0_Instance { S7_SetPoint := 'True'} : TOF_TIME;
      "INT TO REAL" : Real;
   END_VAR
   VAR CONSTANT
      "0" : Int := 0;
      "1" : Int := 1;
   END_VAR
BEGIN

REGION Network 1
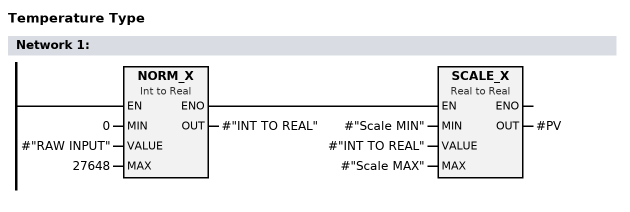
   RUNG wire#powerrail
      { S7_Templates := "[SrcType := Int, DestType := Real]" } Normalize(min := 0, value := #"RAW INPUT", max := 27648, out => #"INT TO REAL")
      { S7_Templates := "[SrcType := Real, DestType := Real]" } Scale(min := #"Scale MIN", value := #"INT TO REAL", max := #"Scale MAX", out => #PV)
   END_RUNG
   // the same network as SCL:
   #"INT TO REAL" := NORM_X(MIN := 0, VALUE := #"RAW INPUT", MAX := 27648);
   #PV := SCALE_X(MIN := #"Scale MIN", VALUE := #"INT TO REAL", MAX := #"Scale MAX");
END_REGION
END_FUNCTION_BLOCK

FUNCTION_BLOCK "Temperature_Control"   // FB3, LAD
{ S7_Optimized_Access := 'TRUE' }
// stored: MemoryReserve 100, SetENOAutomatically false
   VAR_INPUT
      Enable : Bool;
      Man_Enable { ExternalAccessible := 'False'; ExternalVisible := 'False'; ExternalWritable := 'False'} : Bool;
      "Temperature Sensor" : Real;
      "Process Values" : Array[0..1] of Real;
      "Simmer offset" : Real;
      "steam mode" : Int;
      "Setpoint Temperature" : Real;
      "hold time" : Time;
      "Enable temperature Hold" : Bool;
      "manual SP" : Real;
      Jacket : Bool;
   END_VAR
   VAR_OUTPUT
      "Main Valve" : Bool;
      "Simmer Valve" : Bool;
      "Stage Completed" : Bool;
      Running : Bool;
      "Enable Valve" : Bool;
      "Holding Temperature" : Bool;
      "runtime Remaining" : Real;
      "HMI Set Runtime" : Time;
      "HMI Remaining Runtime" : Time;
   END_VAR
   VAR
      "Main Valve SP" : Real;
      "Main Valve SP Reached" : Bool;
      IEC_Timer_0_Instance { S7_SetPoint := 'True'} : TON_TIME;
      IEC_Timer_0_Instance_1 { S7_SetPoint := 'True'} : TON_TIME;
      "Hold Time Completed" : Bool;
      "Reming Time" : DInt;
      Conv_Runtime : Real;
      Runtime : DInt;
      Conv_Runtime2 : Real;
      Remaingtime_1 : Real;
      Remaingtime_2 : Real;
      IEC_Timer_0_Instance_2 { S7_SetPoint := 'True'} : TON_TIME;
      "Main Valve SP Reset" { S7_SetPoint := 'True'} : Real;
      "simmer temperature" : Real;
   END_VAR
   VAR_TEMP   // added for the SCL form of the ladder/FBD networks
      _w1 : Bool;
      _w2 : Bool;
   END_VAR
BEGIN

REGION Network 1
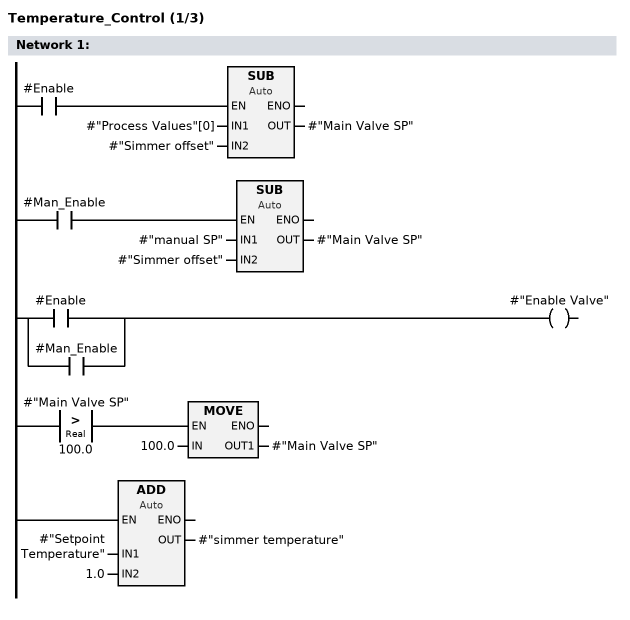
   RUNG wire#powerrail
      Contact( #Enable )
      Sub(in1 := #"Process Values"[0], in2 := #"Simmer offset", out => #"Main Valve SP")
   END_RUNG
   RUNG wire#powerrail
      Contact( #Man_Enable )
      Sub(in1 := #"manual SP", in2 := #"Simmer offset", out => #"Main Valve SP")
   END_RUNG
   RUNG wire#powerrail
      Contact( #Enable )
      wire#w1
      Coil( #"Enable Valve" )
   END_RUNG
   RUNG wire#powerrail
      Contact( #Man_Enable )
   END_RUNG wire#w1
   RUNG wire#powerrail
      { S7_Templates := "SrcType := Real" } GT_Contact(in1 := #"Main Valve SP", in2 := 100.0)
      Move(in := 100.0, out1 => #"Main Valve SP")
   END_RUNG
   RUNG wire#powerrail
      Add(in1 := #"Setpoint Temperature", in2 := 1.0, out => #"simmer temperature")
   END_RUNG
   // the same network as SCL:
   IF #Enable THEN #"Main Valve SP" := #"Process Values"[0] - #"Simmer offset"; END_IF;
   IF #Man_Enable THEN #"Main Valve SP" := #"manual SP" - #"Simmer offset"; END_IF;
   #"Enable Valve" := #Enable OR #Man_Enable;
   IF #"Main Valve SP" > 100.0 THEN #"Main Valve SP" := 100.0; END_IF;
   #"simmer temperature" := #"Setpoint Temperature" + 1.0;
END_REGION

REGION Network 2
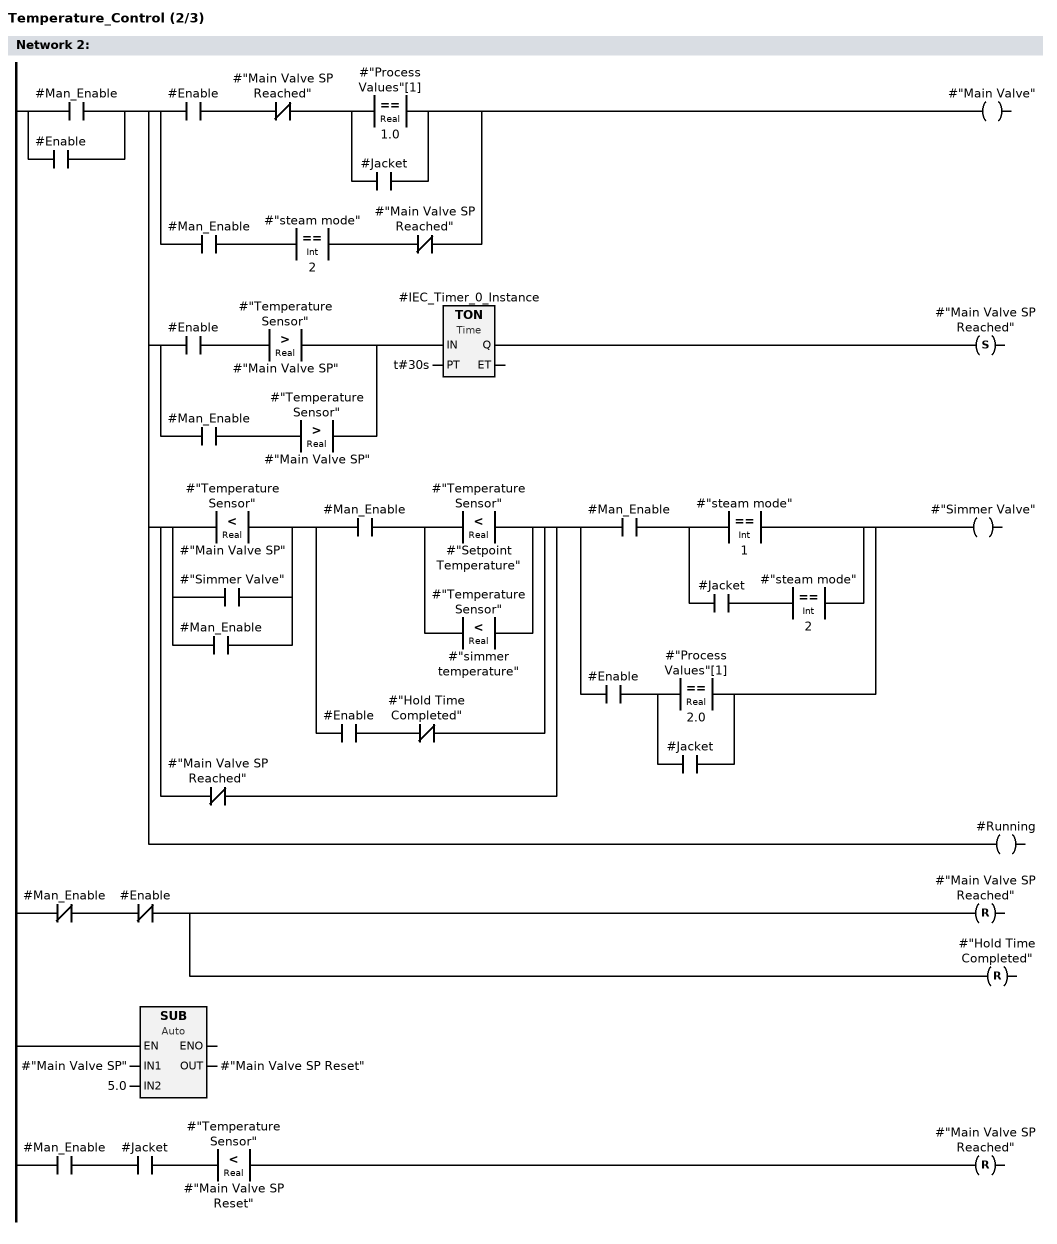
   RUNG wire#powerrail
      Contact( #Man_Enable )
      wire#w1
      Contact( #Enable )
      I_Contact( #"Main Valve SP Reached" )
      wire#w2
      { S7_Templates := "SrcType := Real" } EQ_Contact(in1 := #"Process Values"[1], in2 := 1.0)
      wire#w3
      Coil( #"Main Valve" )
   END_RUNG
   RUNG wire#powerrail
      Contact( #Enable )
   END_RUNG wire#w1
   RUNG wire#w2
      Contact( #Jacket )
   END_RUNG wire#w3
   RUNG wire#w1
      Contact( #Man_Enable )
      { S7_Templates := "SrcType := Int" } EQ_Contact(in1 := #"steam mode", in2 := 2)
      I_Contact( #"Main Valve SP Reached" )
   END_RUNG wire#w3
   RUNG wire#w1
      Contact( #Enable )
      { S7_Templates := "SrcType := Real" } GT_Contact(in1 := #"Temperature Sensor", in2 := #"Main Valve SP")
      wire#w4
      { S7_Templates := "time_type := Time" } #IEC_Timer_0_Instance.TON(pt := t#30s, et =>)
      S_Coil( #"Main Valve SP Reached" )
   END_RUNG
   RUNG wire#w1
      Contact( #Man_Enable )
      { S7_Templates := "SrcType := Real" } GT_Contact(in1 := #"Temperature Sensor", in2 := #"Main Valve SP")
   END_RUNG wire#w4
   RUNG wire#w1
      { S7_Templates := "SrcType := Real" } LT_Contact(in1 := #"Temperature Sensor", in2 := #"Main Valve SP")
      wire#w5
      Contact( #Man_Enable )
      wire#w6
      { S7_Templates := "SrcType := Real" } LT_Contact(in1 := #"Temperature Sensor", in2 := #"Setpoint Temperature")
      wire#w7
      Contact( #Man_Enable )
      wire#w8
      { S7_Templates := "SrcType := Int" } EQ_Contact(in1 := #"steam mode", in2 := 1)
      wire#w9
      Coil( #"Simmer Valve" )
   END_RUNG
   RUNG wire#w1
      Contact( #"Simmer Valve" )
   END_RUNG wire#w5
   RUNG wire#w1
      Contact( #Man_Enable )
   END_RUNG wire#w5
   RUNG wire#w6
      { S7_Templates := "SrcType := Real" } LT_Contact(in1 := #"Temperature Sensor", in2 := #"simmer temperature")
   END_RUNG wire#w7
   RUNG wire#w5
      Contact( #Enable )
      I_Contact( #"Hold Time Completed" )
   END_RUNG wire#w7
   RUNG wire#w1
      I_Contact( #"Main Valve SP Reached" )
   END_RUNG wire#w7
   RUNG wire#w8
      Contact( #Jacket )
      { S7_Templates := "SrcType := Int" } EQ_Contact(in1 := #"steam mode", in2 := 2)
   END_RUNG wire#w9
   RUNG wire#w7
      Contact( #Enable )
      wire#w10
      { S7_Templates := "SrcType := Real" } EQ_Contact(in1 := #"Process Values"[1], in2 := 2.0)
   END_RUNG wire#w9
   RUNG wire#w10
      Contact( #Jacket )
   END_RUNG wire#w9
   RUNG wire#w1
      Coil( #Running )
   END_RUNG
   RUNG wire#powerrail
      I_Contact( #Man_Enable )
      I_Contact( #Enable )
      wire#w11
      R_Coil( #"Main Valve SP Reached" )
   END_RUNG
   RUNG wire#w11
      R_Coil( #"Hold Time Completed" )
   END_RUNG
   RUNG wire#powerrail
      Sub(in1 := #"Main Valve SP", in2 := 5.0, out => #"Main Valve SP Reset")
   END_RUNG
   RUNG wire#powerrail
      Contact( #Man_Enable )
      Contact( #Jacket )
      { S7_Templates := "SrcType := Real" } LT_Contact(in1 := #"Temperature Sensor", in2 := #"Main Valve SP Reset")
      R_Coil( #"Main Valve SP Reached" )
   END_RUNG
   // the same network as SCL:
   #_w1 := #Man_Enable OR #Enable;
   #"Main Valve" := #_w1 AND ((#Enable AND NOT #"Main Valve SP Reached" AND ((#"Process Values"[1] = 1.0) OR #Jacket)) OR (#Man_Enable AND (#"steam mode" = 2) AND NOT #"Main Valve SP Reached"));
   #IEC_Timer_0_Instance(IN := #_w1 AND ((#Enable AND (#"Temperature Sensor" > #"Main Valve SP")) OR (#Man_Enable AND (#"Temperature Sensor" > #"Main Valve SP"))),   // TON
                         PT := t#30s);
   IF #IEC_Timer_0_Instance.Q THEN #"Main Valve SP Reached" := TRUE; END_IF;
   #"Simmer Valve" := #_w1 AND ((((#"Temperature Sensor" < #"Main Valve SP") OR #"Simmer Valve" OR #Man_Enable) AND ((#Man_Enable AND ((#"Temperature Sensor" < #"Setpoint Temperature") OR (#"Temperature Sensor" < #"simmer temperature"))) OR (#Enable AND NOT #"Hold Time Completed"))) OR NOT #"Main Valve SP Reached") AND ((#Man_Enable AND ((#"steam mode" = 1) OR (#Jacket AND (#"steam mode" = 2)))) OR (#Enable AND ((#"Process Values"[1] = 2.0) OR #Jacket)));
   #Running := #_w1;
   IF NOT #Man_Enable AND NOT #Enable THEN
       #"Main Valve SP Reached" := FALSE;
       #"Hold Time Completed" := FALSE;
   END_IF;
   #"Main Valve SP Reset" := #"Main Valve SP" - 5.0;
   IF #Man_Enable AND #Jacket AND (#"Temperature Sensor" < #"Main Valve SP Reset") THEN
       #"Main Valve SP Reached" := FALSE;
   END_IF;
END_REGION

REGION Network 3
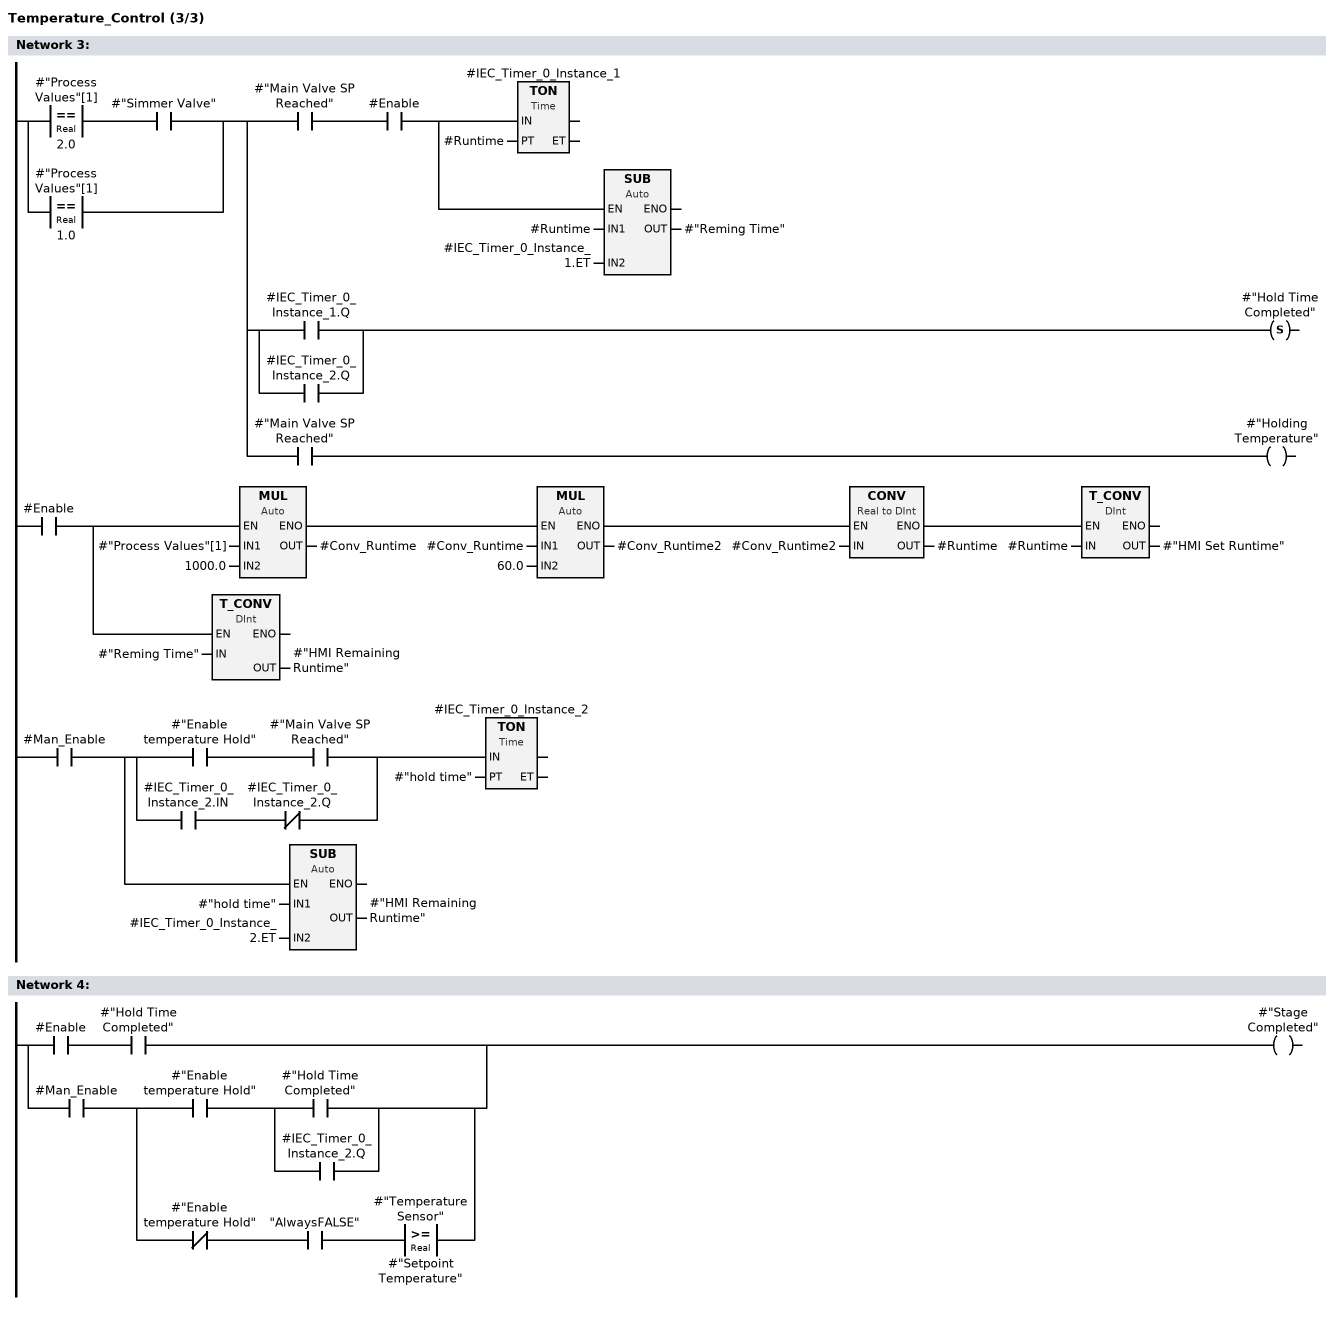
   RUNG wire#powerrail
      { S7_Templates := "SrcType := Real" } EQ_Contact(in1 := #"Process Values"[1], in2 := 2.0)
      Contact( #"Simmer Valve" )
      wire#w1
      Contact( #"Main Valve SP Reached" )
      Contact( #Enable )
      wire#w2
      { S7_Templates := "time_type := Time" } #IEC_Timer_0_Instance_1.TON(pt := #Runtime, et =>)
   END_RUNG
   RUNG wire#powerrail
      { S7_Templates := "SrcType := Real" } EQ_Contact(in1 := #"Process Values"[1], in2 := 1.0)
   END_RUNG wire#w1
   RUNG wire#w2
      Sub(in1 := #Runtime, in2 := #IEC_Timer_0_Instance_1.ET, out => #"Reming Time")
   END_RUNG
   RUNG wire#w1
      Contact( #IEC_Timer_0_Instance_1.Q )
      wire#w3
      S_Coil( #"Hold Time Completed" )
   END_RUNG
   RUNG wire#w1
      Contact( #IEC_Timer_0_Instance_2.Q )
   END_RUNG wire#w3
   RUNG wire#w1
      Contact( #"Main Valve SP Reached" )
      Coil( #"Holding Temperature" )
   END_RUNG
   RUNG wire#powerrail
      Contact( #Enable )
      wire#w4
      Mul(in1 := #"Process Values"[1], in2 := 1000.0, out => #Conv_Runtime)
      Mul(in1 := #Conv_Runtime, in2 := 60.0, out => #Conv_Runtime2)
      { S7_Templates := "[SrcType := Real, DestType := DInt]" } Convert(in := #Conv_Runtime2, out => #Runtime)
      { S7_Templates := "[src_type := DInt, dest_type := Time]" } T_CONV(IN := #Runtime, OUT => #"HMI Set Runtime")
   END_RUNG
   RUNG wire#w4
      { S7_Templates := "[src_type := DInt, dest_type := Time]" } T_CONV(IN := #"Reming Time", OUT => #"HMI Remaining Runtime")
   END_RUNG
   RUNG wire#powerrail
      Contact( #Man_Enable )
      wire#w5
      Contact( #"Enable temperature Hold" )
      Contact( #"Main Valve SP Reached" )
      wire#w6
      { S7_Templates := "time_type := Time" } #IEC_Timer_0_Instance_2.TON(pt := #"hold time", et =>)
   END_RUNG
   RUNG wire#w5
      Contact( #IEC_Timer_0_Instance_2.IN )
      I_Contact( #IEC_Timer_0_Instance_2.Q )
   END_RUNG wire#w6
   RUNG wire#w5
      Sub(in1 := #"hold time", in2 := #IEC_Timer_0_Instance_2.ET, out => #"HMI Remaining Runtime")
   END_RUNG
   // the same network as SCL:
   #_w1 := ((#"Process Values"[1] = 2.0) AND #"Simmer Valve") OR (#"Process Values"[1] = 1.0);
   #_w2 := #_w1 AND #"Main Valve SP Reached" AND #Enable;
   #IEC_Timer_0_Instance_1(IN := #_w2, PT := #Runtime);   // TON
   IF #_w2 THEN #"Reming Time" := #Runtime - #IEC_Timer_0_Instance_1.ET; END_IF;
   IF #_w1 AND (#IEC_Timer_0_Instance_1.Q OR #IEC_Timer_0_Instance_2.Q) THEN
       #"Hold Time Completed" := TRUE;
   END_IF;
   #"Holding Temperature" := #_w1 AND #"Main Valve SP Reached";
   IF #Enable THEN
       #Conv_Runtime := #"Process Values"[1] * 1000.0;
       #Conv_Runtime2 := #Conv_Runtime * 60.0;
       #Runtime := REAL_TO_DINT(#Conv_Runtime2);
       T_CONV(IN := #Runtime, OUT => #"HMI Set Runtime");
       T_CONV(IN := #"Reming Time", OUT => #"HMI Remaining Runtime");
   END_IF;
   #IEC_Timer_0_Instance_2(IN := #Man_Enable AND ((#"Enable temperature Hold" AND #"Main Valve SP Reached") OR (#IEC_Timer_0_Instance_2.IN AND NOT #IEC_Timer_0_Instance_2.Q)),   // TON
                           PT := #"hold time");
   IF #Man_Enable THEN #"HMI Remaining Runtime" := #"hold time" - #IEC_Timer_0_Instance_2.ET; END_IF;
END_REGION

REGION Network 4
   RUNG wire#powerrail
      Contact( #Enable )
      Contact( #"Hold Time Completed" )
      wire#w1
      Coil( #"Stage Completed" )
   END_RUNG
   RUNG wire#powerrail
      Contact( #Man_Enable )
      wire#w2
      Contact( #"Enable temperature Hold" )
      wire#w3
      Contact( #"Hold Time Completed" )
   END_RUNG wire#w1
   RUNG wire#w3
      Contact( #IEC_Timer_0_Instance_2.Q )
   END_RUNG wire#w1
   RUNG wire#w2
      I_Contact( #"Enable temperature Hold" )
      Contact( "AlwaysFALSE" )
      { S7_Templates := "SrcType := Real" } GE_Contact(in1 := #"Temperature Sensor", in2 := #"Setpoint Temperature")
   END_RUNG wire#w1
   // the same network as SCL:
   #"Stage Completed" := (#Enable AND #"Hold Time Completed") OR (#Man_Enable AND ((#"Enable temperature Hold" AND (#"Hold Time Completed" OR #IEC_Timer_0_Instance_2.Q)) OR (NOT #"Enable temperature Hold" AND "AlwaysFALSE" AND (#"Temperature Sensor" >= #"Setpoint Temperature"))));
END_REGION
END_FUNCTION_BLOCK

FUNCTION_BLOCK "Temperature_Control_Concurant"   // FB19, LAD
{ S7_Optimized_Access := 'TRUE' }
// stored: MemoryReserve 100, SetENOAutomatically false
   VAR_INPUT
      Enable : Bool;
      "Temperature Sensor" : Real;
      "Process Values" : Array[0..1] of Real;
      "Main Valve Max Temperature" : Real;
      "simmer offset" : Real;
      "Jacket or Lance" : Bool;
      "auto Run EN" : Bool;
   END_VAR
   VAR_OUTPUT
      "Main Valve" : Bool;
      "Simmer Valve" : Bool;
      Running : Bool;
      "Enable Valve" : Bool;
      "Holding Temperature" : Bool;
      "Run Constant" : Bool;
      "Step Completed" : Bool;
   END_VAR
   VAR
      "Main Valve SP" : Real;
      "Main Valve SP Reached" : Bool;
      IEC_Timer_0_Instance { S7_SetPoint := 'True'} : TON_TIME;
      IEC_Timer_0_Instance_1 { S7_SetPoint := 'True'} : TON_TIME;
   END_VAR
BEGIN

REGION Network 1
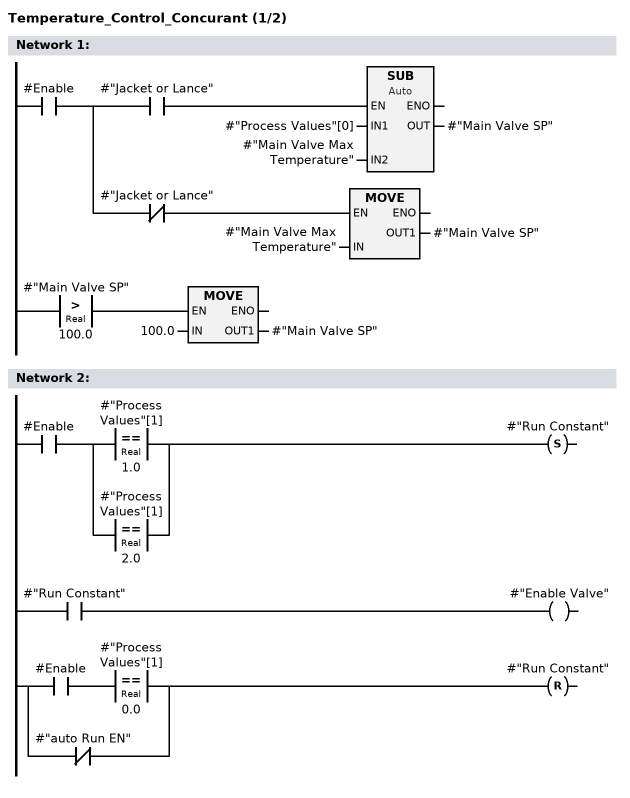
   RUNG wire#powerrail
      Contact( #Enable )
      wire#w1
      Contact( #"Jacket or Lance" )
      Sub(in1 := #"Process Values"[0], in2 := #"Main Valve Max Temperature", out => #"Main Valve SP")
   END_RUNG
   RUNG wire#w1
      I_Contact( #"Jacket or Lance" )
      Move(in := #"Main Valve Max Temperature", out1 => #"Main Valve SP")
   END_RUNG
   RUNG wire#powerrail
      { S7_Templates := "SrcType := Real" } GT_Contact(in1 := #"Main Valve SP", in2 := 100.0)
      Move(in := 100.0, out1 => #"Main Valve SP")
   END_RUNG
   // the same network as SCL:
   IF #Enable AND #"Jacket or Lance" THEN
       #"Main Valve SP" := #"Process Values"[0] - #"Main Valve Max Temperature";
   END_IF;
   IF #Enable AND NOT #"Jacket or Lance" THEN #"Main Valve SP" := #"Main Valve Max Temperature"; END_IF;
   IF #"Main Valve SP" > 100.0 THEN #"Main Valve SP" := 100.0; END_IF;
END_REGION

REGION Network 2
   RUNG wire#powerrail
      Contact( #Enable )
      wire#w1
      { S7_Templates := "SrcType := Real" } EQ_Contact(in1 := #"Process Values"[1], in2 := 1.0)
      wire#w2
      S_Coil( #"Run Constant" )
   END_RUNG
   RUNG wire#w1
      { S7_Templates := "SrcType := Real" } EQ_Contact(in1 := #"Process Values"[1], in2 := 2.0)
   END_RUNG wire#w2
   RUNG wire#powerrail
      Contact( #"Run Constant" )
      Coil( #"Enable Valve" )
   END_RUNG
   RUNG wire#powerrail
      Contact( #Enable )
      { S7_Templates := "SrcType := Real" } EQ_Contact(in1 := #"Process Values"[1], in2 := 0.0)
      wire#w3
      R_Coil( #"Run Constant" )
   END_RUNG
   RUNG wire#powerrail
      I_Contact( #"auto Run EN" )
   END_RUNG wire#w3
   // the same network as SCL:
   IF #Enable AND ((#"Process Values"[1] = 1.0) OR (#"Process Values"[1] = 2.0)) THEN
       #"Run Constant" := TRUE;
   END_IF;
   #"Enable Valve" := #"Run Constant";
   IF (#Enable AND (#"Process Values"[1] = 0.0)) OR NOT #"auto Run EN" THEN #"Run Constant" := FALSE; END_IF;
END_REGION

REGION Network 3
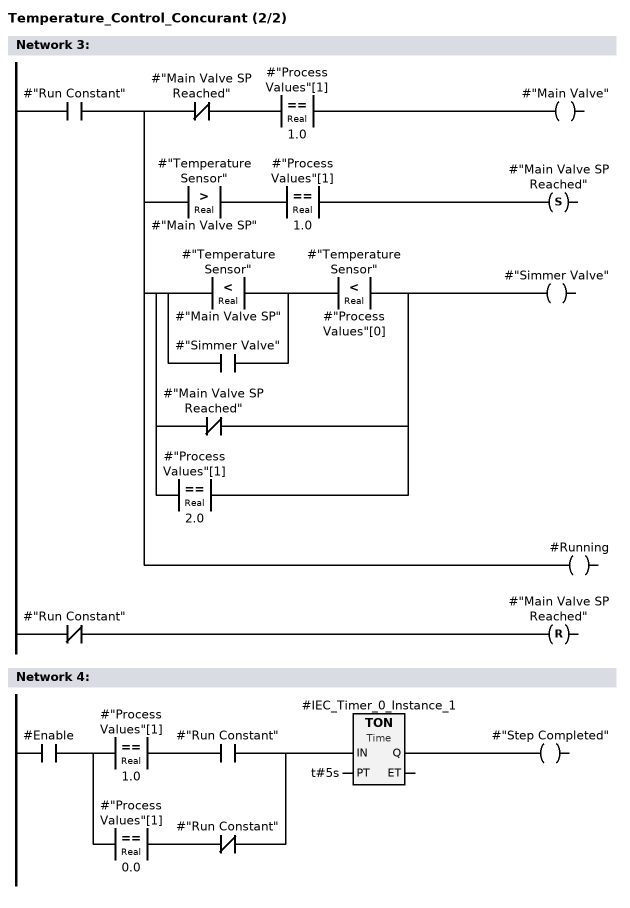
   RUNG wire#powerrail
      Contact( #"Run Constant" )
      wire#w1
      I_Contact( #"Main Valve SP Reached" )
      { S7_Templates := "SrcType := Real" } EQ_Contact(in1 := #"Process Values"[1], in2 := 1.0)
      Coil( #"Main Valve" )
   END_RUNG
   RUNG wire#w1
      { S7_Templates := "SrcType := Real" } GT_Contact(in1 := #"Temperature Sensor", in2 := #"Main Valve SP")
      { S7_Templates := "SrcType := Real" } EQ_Contact(in1 := #"Process Values"[1], in2 := 1.0)
      S_Coil( #"Main Valve SP Reached" )
   END_RUNG
   RUNG wire#w1
      { S7_Templates := "SrcType := Real" } LT_Contact(in1 := #"Temperature Sensor", in2 := #"Main Valve SP")
      wire#w2
      { S7_Templates := "SrcType := Real" } LT_Contact(in1 := #"Temperature Sensor", in2 := #"Process Values"[0])
      wire#w3
      Coil( #"Simmer Valve" )
   END_RUNG
   RUNG wire#w1
      Contact( #"Simmer Valve" )
   END_RUNG wire#w2
   RUNG wire#w1
      I_Contact( #"Main Valve SP Reached" )
   END_RUNG wire#w3
   RUNG wire#w1
      { S7_Templates := "SrcType := Real" } EQ_Contact(in1 := #"Process Values"[1], in2 := 2.0)
   END_RUNG wire#w3
   RUNG wire#w1
      Coil( #Running )
   END_RUNG
   RUNG wire#powerrail
      I_Contact( #"Run Constant" )
      R_Coil( #"Main Valve SP Reached" )
   END_RUNG
   // the same network as SCL:
   #"Main Valve" := #"Run Constant" AND NOT #"Main Valve SP Reached" AND (#"Process Values"[1] = 1.0);
   IF #"Run Constant" AND (#"Temperature Sensor" > #"Main Valve SP") AND (#"Process Values"[1] = 1.0) THEN
       #"Main Valve SP Reached" := TRUE;
   END_IF;
   #"Simmer Valve" := #"Run Constant" AND ((((#"Temperature Sensor" < #"Main Valve SP") OR #"Simmer Valve") AND (#"Temperature Sensor" < #"Process Values"[0])) OR NOT #"Main Valve SP Reached" OR (#"Process Values"[1] = 2.0));
   #Running := #"Run Constant";
   IF NOT #"Run Constant" THEN #"Main Valve SP Reached" := FALSE; END_IF;
END_REGION

REGION Network 4
   RUNG wire#powerrail
      Contact( #Enable )
      wire#w1
      { S7_Templates := "SrcType := Real" } EQ_Contact(in1 := #"Process Values"[1], in2 := 1.0)
      Contact( #"Run Constant" )
      wire#w2
      { S7_Templates := "time_type := Time" } #IEC_Timer_0_Instance_1.TON(pt := t#5s, et =>)
      Coil( #"Step Completed" )
   END_RUNG
   RUNG wire#w1
      { S7_Templates := "SrcType := Real" } EQ_Contact(in1 := #"Process Values"[1], in2 := 0.0)
      I_Contact( #"Run Constant" )
   END_RUNG wire#w2
   // the same network as SCL:
   #IEC_Timer_0_Instance_1(IN := #Enable AND (((#"Process Values"[1] = 1.0) AND #"Run Constant") OR ((#"Process Values"[1] = 0.0) AND NOT #"Run Constant")),   // TON
                           PT := t#5s);
   #"Step Completed" := #IEC_Timer_0_Instance_1.Q;
END_REGION
END_FUNCTION_BLOCK

DATA_BLOCK "Alarms_DB"   // DB2
// stored: InstanceOfName Alarms, InstanceOfType FB
"Alarms"
BEGIN
END_DATA_BLOCK

DATA_BLOCK "GBL_TandD_DB"   // DB104
// stored: InstanceOfName GBL_TandD, InstanceOfType FB
"GBL_TandD"
BEGIN
END_DATA_BLOCK

DATA_BLOCK "Main Control_DB"   // DB1
// stored: InstanceOfName Main Control, InstanceOfType FB
"Main Control"
BEGIN
END_DATA_BLOCK

DATA_BLOCK "FmControl_DB"   // DB26
// stored: InstanceOfName FmControl, InstanceOfType FB
"FmControl"
BEGIN
END_DATA_BLOCK

DATA_BLOCK "Temperature Type_DB_1"   // DB11
// stored: InstanceOfName Temperature Type, InstanceOfType FB
"Temperature Type"
BEGIN
END_DATA_BLOCK

DATA_BLOCK "Temperature Type_DB_2"   // DB12
// stored: InstanceOfName Temperature Type, InstanceOfType FB
"Temperature Type"
BEGIN
END_DATA_BLOCK

DATA_BLOCK "SINA_SPEED_TLG352_DB"   // DB37
AUTHOR : SIEMENS
FAMILY : DRIVES
NAME : SINA_SPD_TLG352
VERSION : 1.0
// stored: InstanceOfName SINA_SPEED_TLG352, InstanceOfType FB
"SINA_SPEED_TLG352"
BEGIN
END_DATA_BLOCK

DATA_BLOCK "BufferMinLevelDebounce"   // DB34
{ S7_Optimized_Access := 'TRUE' }
// stored: InstanceOfName IEC_TIMER, OfSystemLibElement IEC_TIMER, OfSystemLibVersion 1.0
"IEC_TIMER"
   // VAR
   //    PT : Time;
   //    ET { ExternalWritable := 'False'} : Time;
   //    IN : Bool;
   //    Q { ExternalWritable := 'False'} : Bool;
   // END_VAR
BEGIN
END_DATA_BLOCK

DATA_BLOCK "BufferSPLevelDebounce"   // DB35
{ S7_Optimized_Access := 'TRUE' }
// stored: InstanceOfName IEC_TIMER, OfSystemLibElement IEC_TIMER, OfSystemLibVersion 1.0
"IEC_TIMER"
   // VAR
   //    PT : Time;
   //    ET { ExternalWritable := 'False'} : Time;
   //    IN : Bool;
   //    Q { ExternalWritable := 'False'} : Bool;
   // END_VAR
BEGIN
END_DATA_BLOCK

DATA_BLOCK "CoolOverRunTimer"   // DB9
{ S7_Optimized_Access := 'TRUE' }
// stored: InstanceOfName IEC_TIMER, OfSystemLibElement IEC_TIMER, OfSystemLibVersion 1.0
"IEC_TIMER"
   // VAR
   //    PT : Time;
   //    ET { ExternalWritable := 'False'} : Time;
   //    IN : Bool;
   //    Q { ExternalWritable := 'False'} : Bool;
   // END_VAR
BEGIN
END_DATA_BLOCK

DATA_BLOCK "HMI Timer"   // DB38
{ S7_Optimized_Access := 'TRUE' }
// stored: InstanceOfName IEC_TIMER, OfSystemLibElement IEC_TIMER, OfSystemLibVersion 1.0
"IEC_TIMER"
   // VAR
   //    PT : Time;
   //    ET { ExternalWritable := 'False'} : Time;
   //    IN : Bool;
   //    Q { ExternalWritable := 'False'} : Bool;
   // END_VAR
BEGIN
END_DATA_BLOCK

DATA_BLOCK "IEC_Timer_0_DB"   // DB28
{ S7_Optimized_Access := 'TRUE' }
// stored: InstanceOfName IEC_TIMER, OfSystemLibElement IEC_TIMER, OfSystemLibVersion 1.0
"IEC_TIMER"
   // VAR
   //    PT : Time;
   //    ET { ExternalWritable := 'False'} : Time;
   //    IN : Bool;
   //    Q { ExternalWritable := 'False'} : Bool;
   // END_VAR
BEGIN
END_DATA_BLOCK

DATA_BLOCK "IEC_Timer_0_DB_1"   // DB29
{ S7_Optimized_Access := 'TRUE' }
// stored: InstanceOfName IEC_TIMER, OfSystemLibElement IEC_TIMER, OfSystemLibVersion 1.0
"IEC_TIMER"
   // VAR
   //    PT : Time;
   //    ET { ExternalWritable := 'False'} : Time;
   //    IN : Bool;
   //    Q { ExternalWritable := 'False'} : Bool;
   // END_VAR
BEGIN
END_DATA_BLOCK

DATA_BLOCK "IEC_Timer_0_DB_2"   // DB30
{ S7_Optimized_Access := 'TRUE' }
// stored: InstanceOfName IEC_TIMER, OfSystemLibElement IEC_TIMER, OfSystemLibVersion 1.0
"IEC_TIMER"
   // VAR
   //    PT : Time;
   //    ET { ExternalWritable := 'False'} : Time;
   //    IN : Bool;
   //    Q { ExternalWritable := 'False'} : Bool;
   // END_VAR
BEGIN
END_DATA_BLOCK

DATA_BLOCK "IEC_Timer_0_DB_3"   // DB31
{ S7_Optimized_Access := 'TRUE' }
// stored: InstanceOfName IEC_TIMER, OfSystemLibElement IEC_TIMER, OfSystemLibVersion 1.0
"IEC_TIMER"
   // VAR
   //    PT : Time;
   //    ET { ExternalWritable := 'False'} : Time;
   //    IN : Bool;
   //    Q { ExternalWritable := 'False'} : Bool;
   // END_VAR
BEGIN
END_DATA_BLOCK

DATA_BLOCK "IEC_Timer_0_DB_4"   // DB32
{ S7_Optimized_Access := 'TRUE' }
// stored: InstanceOfName IEC_TIMER, OfSystemLibElement IEC_TIMER, OfSystemLibVersion 1.0
"IEC_TIMER"
   // VAR
   //    PT : Time;
   //    ET { ExternalWritable := 'False'} : Time;
   //    IN : Bool;
   //    Q { ExternalWritable := 'False'} : Bool;
   // END_VAR
BEGIN
END_DATA_BLOCK

DATA_BLOCK "IEC_Timer_0_DB_5"   // DB33
{ S7_Optimized_Access := 'TRUE' }
// stored: InstanceOfName IEC_TIMER, OfSystemLibElement IEC_TIMER, OfSystemLibVersion 1.0
"IEC_TIMER"
   // VAR
   //    PT : Time;
   //    ET { ExternalWritable := 'False'} : Time;
   //    IN : Bool;
   //    Q { ExternalWritable := 'False'} : Bool;
   // END_VAR
BEGIN
END_DATA_BLOCK

DATA_BLOCK "IEC_Timer_0_DB_6"   // DB36
{ S7_Optimized_Access := 'TRUE' }
// stored: InstanceOfName IEC_TIMER, OfSystemLibElement IEC_TIMER, OfSystemLibVersion 1.0
"IEC_TIMER"
   // VAR
   //    PT : Time;
   //    ET { ExternalWritable := 'False'} : Time;
   //    IN : Bool;
   //    Q { ExternalWritable := 'False'} : Bool;
   // END_VAR
BEGIN
END_DATA_BLOCK

DATA_BLOCK "IEC_Timer_0_DB_7"   // DB39
{ S7_Optimized_Access := 'TRUE' }
// stored: InstanceOfName IEC_TIMER, OfSystemLibElement IEC_TIMER, OfSystemLibVersion 1.0
"IEC_TIMER"
   // VAR
   //    PT : Time;
   //    ET { ExternalWritable := 'False'} : Time;
   //    IN : Bool;
   //    Q { ExternalWritable := 'False'} : Bool;
   // END_VAR
BEGIN
END_DATA_BLOCK

DATA_BLOCK "OneShotDoseTime"   // DB13
{ S7_Optimized_Access := 'TRUE' }
// stored: InstanceOfName IEC_TIMER, OfSystemLibElement IEC_TIMER, OfSystemLibVersion 1.0
"IEC_TIMER"
   // VAR
   //    PT : Time;
   //    ET { ExternalWritable := 'False'} : Time;
   //    IN : Bool;
   //    Q { ExternalWritable := 'False'} : Bool;
   // END_VAR
BEGIN
END_DATA_BLOCK

DATA_BLOCK "RepeatDoseTimer"   // DB15
{ S7_Optimized_Access := 'TRUE' }
// stored: InstanceOfName IEC_TIMER, OfSystemLibElement IEC_TIMER, OfSystemLibVersion 1.0
"IEC_TIMER"
   // VAR
   //    PT : Time;
   //    ET { ExternalWritable := 'False'} : Time;
   //    IN : Bool;
   //    Q { ExternalWritable := 'False'} : Bool;
   // END_VAR
BEGIN
END_DATA_BLOCK

DATA_BLOCK "UnlatchDoseTimer"   // DB16
{ S7_Optimized_Access := 'TRUE' }
// stored: InstanceOfName IEC_TIMER, OfSystemLibElement IEC_TIMER, OfSystemLibVersion 1.0
"IEC_TIMER"
   // VAR
   //    PT : Time;
   //    ET { ExternalWritable := 'False'} : Time;
   //    IN : Bool;
   //    Q { ExternalWritable := 'False'} : Bool;
   // END_VAR
BEGIN
END_DATA_BLOCK

DATA_BLOCK "logging interval"   // DB27
{ S7_Optimized_Access := 'TRUE' }
// stored: InstanceOfName IEC_TIMER, OfSystemLibElement IEC_TIMER, OfSystemLibVersion 1.0
"IEC_TIMER"
   // VAR
   //    PT : Time;
   //    ET { ExternalWritable := 'False'} : Time;
   //    IN : Bool;
   //    Q { ExternalWritable := 'False'} : Bool;
   // END_VAR
BEGIN
END_DATA_BLOCK

DATA_BLOCK "AN_Scale1"   // DB5
// stored: InstanceOfName An Scaling, InstanceOfType FB
"An Scaling"
BEGIN
END_DATA_BLOCK

DATA_BLOCK "An Scale2"   // DB6
// stored: InstanceOfName An Scaling, InstanceOfType FB
"An Scaling"
BEGIN
END_DATA_BLOCK

DATA_BLOCK "An Scale3"   // DB7
// stored: InstanceOfName An Scaling, InstanceOfType FB
"An Scaling"
BEGIN
END_DATA_BLOCK

DATA_BLOCK "An Scale4"   // DB8
// stored: InstanceOfName An Scaling, InstanceOfType FB
"An Scaling"
BEGIN
END_DATA_BLOCK

DATA_BLOCK "FMDensity Sts"   // DB23
// stored: InstanceOfName FmStsCodes, InstanceOfType FB
"FmStsCodes"
BEGIN
END_DATA_BLOCK

DATA_BLOCK "FMReferenceDensity Sts"   // DB24
// stored: InstanceOfName FmStsCodes, InstanceOfType FB
"FmStsCodes"
BEGIN
END_DATA_BLOCK

DATA_BLOCK "FMTemperature Sts"   // DB25
// stored: InstanceOfName FmStsCodes, InstanceOfType FB
"FmStsCodes"
BEGIN
END_DATA_BLOCK

DATA_BLOCK "FmCorrectedVolumeFlow Sts"   // DB22
// stored: InstanceOfName FmStsCodes, InstanceOfType FB
"FmStsCodes"
BEGIN
END_DATA_BLOCK

DATA_BLOCK "FmVolume Flow STS"   // DB21
// stored: InstanceOfName FmStsCodes, InstanceOfType FB
"FmStsCodes"
BEGIN
END_DATA_BLOCK

DATA_BLOCK "MassFlowDiag"   // DB20
// stored: InstanceOfName FmStsCodes, InstanceOfType FB
"FmStsCodes"
BEGIN
END_DATA_BLOCK

DATA_BLOCK "Liquid_Pump"   // DB10
// stored: InstanceOfName VFD Type, InstanceOfType FB
"VFD Type"
BEGIN
END_DATA_BLOCK

DATA_BLOCK "FlowmeterValve"   // DB19
// stored: InstanceOfName Valve_Type, InstanceOfType FB
"Valve_Type"
BEGIN
END_DATA_BLOCK

DATA_BLOCK "IBCValve"   // DB4
// stored: InstanceOfName Valve_Type, InstanceOfType FB
"Valve_Type"
BEGIN
END_DATA_BLOCK

DATA_BLOCK "PumpValve"   // DB17
// stored: InstanceOfName Valve_Type, InstanceOfType FB
"Valve_Type"
BEGIN
END_DATA_BLOCK

DATA_BLOCK "doseValve"   // DB18
// stored: InstanceOfName Valve_Type, InstanceOfType FB
"Valve_Type"
BEGIN
END_DATA_BLOCK
